(* IEC 61131-3 sources: myCodes/Stone/07.02.2022 - OOPs Approach/MPx_One_New/Mpx_One_Source_Code/MPx_One/3. USHPXMPX010A1/USHPXMPX010A1/[8c990d04-4ef8-4ca1-9757-e845a4517aeb]/Application (part 2) *)

(* ---- 060_MainRegMng.st ---- *)
USING Libs.Logics;
USING System.Timer;
USING System;
USING System.Math;
USING System.Util;

// Uncomment to enable day/night logging
//{DEFINE DNLOGS 1}

VAR_GLOBAL
    MstTempRegStatus : BOOL;
END_VAR

NAMESPACE LibraryNamespaceAndVersion

PROGRAM MainRegMng
    VAR

        TP_s_Timed : TP;
        EEVStartSR : SR;

        CleanRF : RF_TRIG;
        CleanTON : TON;
        //CleanTON_R_Trig : R_TRIG;

        //ContStatusRT : R_TRIG;

        DoorTON : TON;
        DoorLigthTON : TON;
        //DoorOnUsed, DoorOffUsed : FctIsUsed;

        DayNightTrigger, CurtainTrigger : RF_TRIG;//, OnOffDinTrigger : RFTrig;
        DayNightScheduler : MPXScheduler;

        StandbyTON, AndTimeoutTON, AlarmONTON, AlarmTON : TON;
        ContCycle_Pulse : TP;
        StandBy_DIN_R_TRIG : R_TRIG;
        Standby_RS : RS;

        DutySetON, DutySetOFF : TON;

        // Generic function
        AlarmFct : ARRAY [1..1] OF libs.GenericFunctionMng.GenFct_Alarm;
        StageFct : ARRAY [1..1] OF Libs.GenericFunctionMng.GenFct_Stage;
        {IF NOT DEF(MPXONE_BASIC)}
        ModulFct : ARRAY [1..1] OF libs.GenericFunctionMng.GenFct_Modulating;
        {ENDIF}

        TempRegHyst_Left, TempRegHyst_Left2 : REAL;
        TempRegHyst_Right, TempRegHyst_Right2 : REAL;
        //SetP_On, SetP_On2 : REAL;
        //SetP_Off, SetP_Off2 : REAL;

        F_EDGE_firstCycle : F_EDGE;
        FirstCicle_L_Trig   : F_TRIG;

    END_VAR

    VAR_TEMP
        //tmpTempSetP_Offs, tmpTempSetP_Offs2 : REAL;
        AirOffBroken_Delta, AirOnBroken_Delta : REAL;
        EEVOpenOk : BOOL;
        i : DINT;
        //tmpDefCondition : BOOL;
        CompFanDelay_TIME : TIME;

        AlarmTime : TIME;
    END_VAR

    //wait restore default
    IF SW_Update THEN
        RETURN;
    END_IF;

    {REGION STARTUP DELAY}
    // Following regulation will be enabled after the startup delay
    F_EDGE_firstCycle(In := firstCycle);
    FirstCicle_L_Trig(CLK := firstCycle);   // TRAC #115: Stop regoulation at startup (first cycle) in case of startup defrost set
    IF firstCycle OR (FirstCicle_L_Trig.Q AND StartupDef)  THEN
        RETURN;
    END_IF;
    {ENDREGION}

    VirtualProbe := (AnalogInputs.Fct.AirOff * TO_REAL(100 - VirtualComposition) + AnalogInputs.Fct.AirOn * TO_REAL(VirtualComposition)) / 100.0;

    {REGION DAY / NIGHT}
    // Default DayStatus value at startup TRUE

    // Align TOD datatype for APPLICA
    FOR i := LOWER_BOUND(TimeBandStart, 1) TO UPPER_BOUND(TimeBandStart, 1) DO
        ALIGN_TB_TOD(TimeBandStart[i]);
    END_FOR;
    FOR i := LOWER_BOUND(TimeBandEnd, 1) TO UPPER_BOUND(TimeBandEnd, 1) DO
        ALIGN_TB_TOD(TimeBandEnd[i]);
    END_FOR;

    DayNightScheduler(
        CurrentDT := CurrDateTime, Today := CurrentDoW,
        StartTB := TimeBandStart,
        StopTB := TimeBandEnd);

    IF DayNightScheduler.StartTrigger THEN
        DayStatus := TRUE;
    END_IF;

    IF DayNightScheduler.StopTrigger THEN
        DayStatus := FALSE;
    END_IF;

    // Check the curtain switch input
    CurtainTrigger(CLK := DigitalInputs.Fct.Curtain);
    IF CurtainTrigger.Q THEN
        DayStatus := DigitalInputs.Fct.Curtain;
    END_IF;

    // Light adjustment
    DayNightTrigger(CLK := DayStatus);
    IF DayNightTrigger.Q AND Dout_Cfg.Fct.Light.Ch > 0 THEN
        LightsOn := DayStatus;
    END_IF;

    // Light management when door switch is configured
    IF DoorTrigger.Q AND Dout_Cfg.Fct.Light.Ch > 0 THEN
        IF DigitalInputs.Fct.DoorOn OR DigitalInputs.Fct.DoorOff THEN
            LightsOn := DigitalInputs.Fct.DoorOn OR DigitalInputs.Fct.DoorOff;
        ELSIF LightOnDoorDelay = 0 THEN
            LightsOn := FALSE;
        END_IF;
    END_IF;

    // Door timeout for light mng

    DoorLigthTON(IN := LightsOn AND Dout_Cfg.Fct.Light.Ch > 0 AND
        NOT ((DigitalInputs.Fct.DoorOn AND Din_Cfg.fct.DoorOn.Ch > 0) OR (DigitalInputs.Fct.DoorOff AND Din_Cfg.fct.DoorOff.Ch > 0)),
        PT := TO_TIME(TO_DINT(LightOnDoorDelay) * 60 * 1000));

    IF DoorLigthTON.Q AND (Din_Cfg.fct.DoorOff.Ch > 0 OR Din_Cfg.fct.DoorOn.Ch > 0) THEN
        LightsOn := FALSE;
    END_IF;

    // Master / Slave sync
    IF isMaster THEN
        // Notify the slaves on master light status
        FOR i := 1 TO TO_DINT(SlavesNum) DO
            {IF NOT DEF(MPXONE_BASIC)}
            Slaves[i].myCoilStatus[089] := LightsOn;    // set NetworkLight
            Slaves[i].myCoilStatus[079] := AuxOn;       // set NetworkAux
            {ELSE}
            Slaves[i].myCoilStatus[080] := LightsOn;    // set NetworkLight
            Slaves[i].myCoilStatus[071] := AuxOn;       // set NetworkAux
            {ENDIF}
        END_FOR;
    END_IF;

    // Auxiliary output
    CASE CmdAux OF
        0: AuxOn := FALSE;
        1: AuxOn := DayNightOutput AND DayStatus;
        2: AuxOn := TRUE;
    END_CASE;

    {ENDREGION}
    {REGION TIMER FUNCTION}
    TP_s_Timed(IN := DigitalInputs.Fct.Timed, PT := TO_TIME(TO_UINT(TimerDelay) * 60 * 1000));
    TimedOn := TP_s_Timed.Q;
    {ENDREGION}

    {REGION TEMPERATURE REGULATION}
    // regulation probe selection
    RegProbe := VirtualProbe;

    // Night regulation with return temperature probe
    IF NOT DayStatus AND NightPrbReg THEN
        RegProbe := AnalogInputs.Fct.AirOn;
    END_IF;

    // Check setpoint limits on parameter
    TempSetP := MAX(MinTempSet, TempSetP);
    TempSetP := MIN(MaxTempSet, TempSetP);

    TempSetP2 := MAX(MinTempSet, TempSetP2);
    TempSetP2 := MIN(MaxTempSet, TempSetP2);

   //23/01/2020 Filippo Pizzo - TRAC #99: changed action from trigger to keep forced the unit off by remote off

    // Din remote ON/OFF --> force unit off
//    IF DigitalInputs.Fct.RemoteOff THEN
//        UnitStatus := FALSE;
//    END_IF;
    /*
    OnOffDinTrigger(In := DigitalInputs.Fct.RemoteOff);
    IF OnOffDinTrigger.Out THEN
        UnitStatus := NOT DigitalInputs.Fct.RemoteOff;
    END_IF;
    */

    IF UnitOn AND NOT WaitForUpdate THEN
        // Regulation not in alarm
        IF NOT Alarms.Al.AlExtDin.Info.Active AND (NOT(Alarms.Al.AlDelayExtDin.Info.Active AND AlDinDelay>0)) //TRAC #111: if AlDinDelay (param.DIb) = 0 --> only warning
                AND NOT GenFctAlarm_Serious THEN //ISSUE #35

            {REGION TEMPERATURE REGULATION}
            TempRegHyst_Right := TempSetP;
            TempRegHyst_Left := TempSetP;
            TempRegHyst_Right2 := TempSetP2;
            TempRegHyst_Left2 := TempSetP2;

//            SetP_On := TempSetP;
//            SetP_Off := TempSetP;
//            SetP_On2 := TempSetP2;
//            SetP_Off2 := TempSetP2;

            // Control probe lookup
            IF Ain_Cfg.Fct.AirOn.Ch > 0 AND Ain_Cfg.Fct.AirOn.Ch <= TO_SINT(MAX_AIN_CH) THEN
                AirOnBroken := Alarms.Al.Al_PrbBroken[Ain_Cfg.Fct.AirOn.Ch].Info.Active;
            ELSIF Ain_Cfg.Fct.AirOn.Ch < 0 AND Ain_Cfg.Fct.AirOn.Ch >= -4 THEN
                AirOnBroken := Alarms.Al.Al_SerialInputs[-Ain_Cfg.Fct.AirOn.Ch].Info.Active;
            ELSE
                // Probe not configured
                AirOnBroken := TRUE;
            END_IF;

            IF Ain_Cfg.Fct.AirOff.Ch > 0 AND Ain_Cfg.Fct.AirOff.Ch <= TO_SINT(MAX_AIN_CH) THEN

            AirOffBroken := Alarms.Al.Al_PrbBroken[Ain_Cfg.Fct.AirOff.Ch].Info.Active;
            ELSIF Ain_Cfg.Fct.AirOff.Ch < 0 AND Ain_Cfg.Fct.AirOff.Ch >= -4 THEN
                AirOffBroken := Alarms.Al.Al_SerialInputs[-Ain_Cfg.Fct.AirOff.Ch].Info.Active;
            ELSE
                // Probe not configured
                AirOffBroken := TRUE;
            END_IF;

            // Both probe broken or disconnected or not configured
            DutySettings := AirOffBroken AND AirOnBroken;

            // Probe error compensation for AIR OFF broken
            AirOffBroken_Delta := (PrbErrorOffset *  ((100 - TO_REAL(VirtualComposition)) / 100)) * TO_REAL(AirOffBroken);

            // Probe error compensation for AIR ON broken
            AirOnBroken_Delta := (PrbErrorOffset * (TO_REAL( VirtualComposition) / 100)) * TO_REAL(AirOnBroken);

            IF AirOffBroken THEN
                IF VirtualComposition = 0 THEN
                    DutySettings := TRUE;
                ELSE
                     // Switch on other regulation probe
                    RegProbe := AnalogInputs.Fct.AirOn;
                END_IF;
            END_IF;

            IF AirOnBroken THEN
                IF VirtualComposition = 100 THEN
                    DutySettings := TRUE;
                ELSE
                     // Switch on other regulation probe
                    RegProbe := AnalogInputs.Fct.AirOff;
                END_IF;
            END_IF;

            TempRegHyst_Right := TempRegHyst_Right + AirOffBroken_Delta - AirOnBroken_Delta;
            TempRegHyst_Left := TempRegHyst_Left + AirOffBroken_Delta - AirOnBroken_Delta;

            TempRegHyst_Right2 := TempRegHyst_Right2 + AirOffBroken_Delta - AirOnBroken_Delta;
            TempRegHyst_Left2 := TempRegHyst_Left2 + AirOffBroken_Delta - AirOnBroken_Delta;

            IF TempCtrl_DirRev THEN
                                //Standard regulation + Day/Night delta + Smoothline offset + Probe broken offset
                TempRegHyst_Right := TempRegHyst_Right - (SetpNightOffset * TO_REAL( NOT DayStatus ))
                            + (SmLineTempOffset * TO_REAL(EnSmoothLine));
                TempRegHyst_Left := TempRegHyst_Left - TempDiff - (SetpNightOffset * TO_REAL(NOT DayStatus));

                TempRegHyst_Right2 := TempRegHyst_Right2- (SetpNightOffset * TO_REAL( NOT DayStatus ))
                            + (SmLineTempOffset * TO_REAL(EnSmoothLine));

                TempRegHyst_Left2 := TempRegHyst_Left2 - TempDiff2  - (SetpNightOffset * TO_REAL( NOT DayStatus ));

                // Update BMS variables
                ActualTempSetpoint := TempRegHyst_Right;
                ActualTemp2Setpoint := TempRegHyst_Right2;
            ELSE
                //Standard regulation + Day/Night delta + Smoothline offset + Probe broken offset
                TempRegHyst_Right := TempRegHyst_Right + TempDiff + (SetpNightOffset * TO_REAL(NOT DayStatus));
                TempRegHyst_Left := TempRegHyst_Left + (SetpNightOffset * TO_REAL( NOT DayStatus ))
                            - (SmLineTempOffset * TO_REAL(EnSmoothLine));

                TempRegHyst_Right2 := TempRegHyst_Right2 + TempDiff2  + (SetpNightOffset * TO_REAL( NOT DayStatus ));
                TempRegHyst_Left2 := TempRegHyst_Left2 + (SetpNightOffset * TO_REAL( NOT DayStatus ))
                            - (SmLineTempOffset * TO_REAL(EnSmoothLine));

                // Update BMS variables
                ActualTempSetpoint := TempRegHyst_Left;
                ActualTemp2Setpoint := TempRegHyst_Left2;
            END_IF;

            // Double thermostat logic
            IF TempDiff2 > 0.0 THEN

                TempReg(
                	In        := AnalogInputs.Fct.AirOff,
                	SetP      := TempRegHyst_Left,
                	DiffLeft  := 0.0,
                	DiffRight := TempRegHyst_Right - TempRegHyst_Left,
                	Reverse   := TempCtrl_DirRev
                );

                TempReg2(
                	In        := AnalogInputs.Fct.AirOn,
                	SetP      := TempRegHyst_Left2,
                	DiffLeft  := 0.0,
                	DiffRight := TempRegHyst_Right2 - TempRegHyst_Left2,
                	Reverse   := TempCtrl_DirRev
                );
//                TempReg(In := AnalogInputs.Fct.AirOff,
//                    Left := TempRegHyst_Left,
//                    Right := TempRegHyst_Right,
//                    Reverse := TempCtrl_DirRev);

//                TempReg2(In := AnalogInputs.Fct.AirOn,
//                    Left := TempRegHyst_Left2,
//                    Right := TempRegHyst_Right2,
//                    Reverse := TempCtrl_DirRev);

                IF DoubleThermostatConf THEN
                    // OR Condition
                    TempRegStatus := TempReg.Out OR TempReg2.Out;
                    MstTempRegStatus := TempRegStatus;
                ELSE
                    // AND Condition
                    AndTimeoutTON(IN := (TempReg.Out XOR TempReg2.Out) AND DoubleThermSafety > 0, PT := TO_TIME(TO_UINT(DoubleThermSafety) * 60 * 1000));
                        (*Regolation starts if there are request from Sm AND Sr   OR   if there are only one of those AND DoubleThermSafety (dbS) time setted*)
                    TempRegStatus := (TempReg.Out AND TempReg2.Out) OR (AndTimeoutTON.Q AND DoubleThermSafety > 0);
                    MstTempRegStatus := TempRegStatus;
                END_IF;
          ELSE
                TempReg(
                	In        := RegProbe,
                	SetP      := TempRegHyst_Left,
                	DiffLeft  := 0.0,
                	DiffRight := TempRegHyst_Right - TempRegHyst_Left,
                	Reverse   := TempCtrl_DirRev
                );
//                TempReg(In := RegProbe,
//                    Left := TempRegHyst_Left,
//                    Right := TempRegHyst_Right,
//                    Reverse := TempCtrl_DirRev);

                // No double thermostat
                TempRegStatus := TempReg.Out;
                MstTempRegStatus := TempRegStatus;
            END_IF;

            {ENDREGION}

            {REGION CONTINUOUS CYCLE}
            /* Alesssandro Balzan 03/07/2020 changed logic of activation Used TP and added control from disply */

            ContCycle_Pulse(
            	IN := DigitalInputs.Fct.ContCycle OR ManContCycle_byDisplay OR ManContCycle_bySuperv,
            	PT := TO_TIME(TO_DINT(ContCycleTout) * 1000 * 3600)
            );

            IF (DigitalInputs.Fct.ContCycle OR ManContCycle_byDisplay OR ManContCycle_bySuperv) AND ContCycle_Pulse.Q THEN
                ManContinuous := TRUE;
            ELSE
                ContCycle_Pulse(PT := T#0ms); // reset TP
                ManContinuous           := FALSE;
                ManContCycle_byDisplay  := FALSE;
                ManContCycle_bySuperv   := FALSE;
            END_IF;

            //stopped by Alarm
            IF ManContinuous AND ( TempAlarms[1].Low OR TempAlarms[2].Low) AND ContCycleTout > 0 THEN
                ManContinuous           := FALSE;
                ManContCycle_byDisplay  := FALSE;
                ManContCycle_bySuperv   := FALSE;
            END_IF;

            // Defrost priority
            IF ManContinuous AND DfrStatus > DFR_IDLE AND DfrPriorityCont THEN
                ManContinuous           := FALSE;
                ManContCycle_byDisplay  := FALSE;
                ManContCycle_bySuperv   := FALSE;
            END_IF;

            // Keep the regulation active until temperature reach Low temperature alarm threshold
            TempRegStatus := TempRegStatus OR ManContinuous;
            MstTempRegStatus := MstTempRegSTatus OR ManContinuous;

            {ENDREGION}

            {REGION DUTY SETTINGS}
            // Act like a slave for temperature regulation
            IF NOT isMaster AND DutySettings AND NOT Alarms.Al.Al_MA.Info.Active THEN
                TempRegStatus := MstRegStatus;
                RegProbe := MstRegTemp;
                DutySettings := FALSE;
            END_IF;

            IF DutySettings THEN
                DutySetON(IN := NOT DutySetOFF.Q, PT := TO_TIME(TO_DINT(DutySetOnTime) * 60 * 1000));
                DutySetOFF(IN := DutySetON.Q, PT := T#15m);

                TempRegStatus := NOT DutySetON.Q AND NOT DutySetOFF.Q;

                TempRegStatus := TempRegStatus AND DutySetOnTime > 0;

            END_IF;

            // Regulation alarm trigger
            Alarms.Al.Al_Reg.Info.Trigger := DutySettings;
            {ENDREGION}

            {REGION DOOR MANAGEMENT}
            /*DoorOnUsed(FunctionValue := DIN_DOOR_INDEX, Fct := DinFct);
            DoorOffUsed(FunctionValue := DIN_DOOR_ON_INDEX, Fct := DinFct);*/

            DoorTrigger(CLK := DigitalInputs.Fct.DoorOff OR DigitalInputs.Fct.DoorOn);

            Alarms.Al.Warn_Door.Info.Trigger := DigitalInputs.Fct.DoorOff OR DigitalInputs.Fct.DoorOn;

            DoorTON(IN := DigitalInputs.Fct.DoorOff OR DigitalInputs.Fct.DoorOn, PT := TO_TIME(TO_DINT(HighTempBypDoor) * 60 * 1000));
            Alarms.Al.Al_Door.Info.Trigger := DoorTON.Q;

            IF DigitalInputs.Fct.DoorOff AND NOT DoorTON.Q THEN
                TempRegStatus := FALSE;
            END_IF;

//            {IF NOT DEF(MPXONE_BASIC)}
//            myVarTest := FALSE;
//            {ENDIF}

            {ENDREGION}

            {REGION STANDBY}
            StandBy_DIN_R_TRIG(CLK := DigitalInputs.Fct.Standby);
            Standby_RS(S := StandBy_DIN_R_TRIG.Q,
                        R1 := StartupTimeTON.ET > T#0ms OR NOT DigitalInputs.Fct.Standby OR StbyTout = 0);

            Alarms.Al.Status_Standby.Info.Trigger := Standby_RS.Q1 AND NOT StandbyTON.Q;
            StandbyTON(IN := Standby_RS.Q1, PT := TO_TIME(TO_DINT(StbyTout) * 60 * 1000));
            IF Standby_RS.Q1 AND NOT StandbyTON.Q AND StbyTout > 0 THEN
                TempRegStatus := FALSE;
            END_IF;

            {ENDREGION}

            {REGION CLEAN STATUS}
            Alarms.Al.Status_Clean.Info.Trigger := ManClean AND NOT CleanTON.Q;

            CleanRF(CLK := DigitalInputs.Fct.Clean);
            IF CleanRF.Q THEN
                ManClean := DigitalInputs.Fct.Clean;
            END_IF;

            CleanTON(IN := ManClean AND CleanTout > 0, PT := TO_TIME(TO_UDINT(CleanTout) * 60 * 1000));
            IF ManClean AND NOT CleanTON.Q THEN
                TempRegStatus := FALSE;
            END_IF;

            IF (CleanTout > 0 AND CleanTON.ET >= TO_TIME(TO_UDINT(CleanTout) * 60 * 1000)) THEN
                ManClean := FALSE;
            END_IF;

            {ENDREGION}

            // Stop regulation with Natural defrost by running time,
            IF DfrNatural OR DfrCompOff OR           // with compressor=off and defrost until post dripping Ticket TRAC 115)
                (NOT(CompOn) AND DfrStatus>DFR_IDLE AND DfrStatus<DFR_POST_DRIPPING AND DfrType<>1 AND DfrType<>3) THEN

                TempRegStatus := FALSE;

                // Added for hotgas: compON = ON during defrost (not dripping) Independently from request
            ELSIF (DfrType=1 OR DfrType=3) AND DfrStatus>DFR_IDLE AND DfrStatus<DFR_DRIPPING THEN
                TempRegStatus := TRUE;
            END_IF;

            {IF NOT DEF(MPXONE_BASIC)}
            // P10 management
            IF ExvEnCloseLsa AND (Alarms.Al.Al_LSA.Info.Trigger OR Alarms.Al.Al_LSH.Info.Trigger) AND NOT(isMaster AND MstVlvConfig) THEN
                TempRegStatus := FALSE;
//                MstTempRegStatus := FALSE;
            END_IF;
            // PM5 management
            IF ExvEnCloseMOP AND Alarms.Al.Al_MOP.Info.Trigger AND NOT(isMaster AND MstVlvConfig) THEN
                TempRegStatus := FALSE;
//                MstTempRegStatus := FALSE;
            END_IF;
            {ENDIF}

            {REGION Network compressor/solenoid valve output on the Master}
            SlavesTempReq := FALSE;
            // check "TempRegStatus"
            IF isMaster AND SlavesNum > 0 AND MstVlvConfig THEN
                FOR i := 1 TO UPPER_BOUND(Slaves, 1) DO
                    {IF NOT DEF(MPXONE_BASIC)}
                    IF Slaves[i].myInputStatus[87]  THEN
                        SlavesTempReq := TRUE;
                        EXIT;
                    END_IF;
                    {ELSE}
                    IF Slaves[i].myInputStatus[72]  THEN
                        SlavesTempReq := TRUE;
                        EXIT;
                    END_IF;
                    {ENDIF}
                END_FOR;
            END_IF;

            TempRegStatus := TempRegStatus OR SlavesTempReq;
            {ENDREGION}

            {REGION Safety time}
            MinOnT := LIMIT(MinOnT, 0, 15);
            MinOnOnSameT := LIMIT(MinOnOnSameT, 0, 15);
            MinOffT := LIMIT(MinOffT, 0, 15);
            {ENDREGION }

            // Valve has reached the startup opening?
            {IF NOT DEF(MPXONE_BASIC)}
            IF ValveCnf = 6 AND Alarms.Al.Al_Edc.Info.Active THEN
                EEVOpenOk := TRUE;
            ELSE
                EEVOpenOk := (MachineVars.Engine_vars.EEV_vars.CurrentEstimatedPosition > MachineParams.Engine_params.EEV_PARAMS.MinSteps) AND
                            NOT Alarms.Al.Al_Edc.Info.Active;
            END_IF;
            {ELSE}
                EEVOpenOk := TRUE;
            {ENDIF}

            EEVStartSR(
                S1 := TempRegStatus AND (EEVOpenOk OR ValveCnf = 0 OR (isMaster AND SlavesTempReq)),
                R := NOT TempRegStatus
                );

            {REGION Compressor safety times}
            // Comp off during some phase of defrost
            //tmpDefCondition := DfrStatus = DFR_IDLE OR DfrStatus = DFR_POST_DRIPPING ;

            // Allow pump down (NOT AVAILABLE IN CASE OF LIQUID SOLENOID VALVE)
            /*IF DfrPmpDwnDuration > MinOnT THEN
                tmpDefCondition := tmpDefCondition OR DfrStatus = DFR_CALL;
            END_IF;*/

            CntDwnSafT(
                DevReq := EEVStartSR.Q1,
                DevStatus := CompOn,
                MinOnT := MinOnT * 60,
                MinOffT := MinOffT * 60,
                MinOnOnSameT := MinOnOnSameT * 60,
                ResSafT := DfrSafetyTime AND DfrStatus > DFR_CALL,
                DevAlrm := CompAllAlrm,
                En_FB := TRUE

        //        DevOn => BOOL,
        //        FrcdOffByT => ShowCntDwnOff,
        //        FrcdOnByT => ShowCntDwnOn,
        //        CntDwnTSaf => CntDwnT_FrcdOff,
        //        CntDwnTMinOn => CntDwnT_FrcdOn
        //        AbleToOn => BOOL,
        //        AbleToOff => BOOL
                );

            // Function output
            CASE CmdComp OF
                0: // Forced OFF
                    CompOn := FALSE;
                    CompFanDelay_TON(IN := FALSE, PT := T#0ms);
                1: // Automatic
                    IF CompFanDelay > 0 THEN
                        CompFanDelay_TIME := TO_TIME(TO_UDINT(CompFanDelay) * 60 * 1000);
                        CompFanDelay_TON();
                        IF F_EDGE_firstCycle.Out AND CntDwnSafT.DevOn THEN
                            F_EDGE_firstCycle.Reset := TRUE;
                            CompFanDelay_TON(IN := TRUE, PT := CompFanDelay_TIME);
                        ELSIF NOT (CompFanDelay_TON.ET > T#0ms) THEN
                            CompOn := CntDwnSafT.DevOn;
                        ELSIF CompFanDelay_TON.ET >= CompFanDelay_TIME THEN
                            CompFanDelay_TON(IN := FALSE, PT := T#0ms);
                        END_IF;
                    ELSE
                        CompOn := CntDwnSafT.DevOn;
                    END_IF;
                2: // Forced ON
                    CompOn := TRUE;
                    CompFanDelay_TON(IN := FALSE, PT := T#0ms);
            END_CASE;

            // Align slaves about current regulation status
            IF isMaster THEN
                FOR i:=1 TO TO_DINT(SlavesNum) DO
                    {IF NOT DEF(MPXONE_BASIC)}
                    Slaves[i].myCoilStatus[77] := CompOn;   //Set MstRegStatus
                    Slaves[i].myHoldingRegisters[239] := TO_UINT(RegProbe * 10); //Set MstRegTemp
                    {ELSE}
                    Slaves[i].myCoilStatus[069] := CompOn;  //Set MstRegStatus
                    Slaves[i].myHoldingRegisters[178] := TO_UINT(RegProbe * 10); //Set MstRegTemp
                    {ENDIF}
                END_FOR;
            END_IF;
            {ENDREGION }
        ELSE
            // Regulation in alarm with A10 config
            AlarmTime := TO_TIME(TO_REAL(CmpAlConfig) / 100.0 * 15 * 60 * 1000);

            AlarmONTON(IN := NOT AlarmTON.Q, PT := AlarmTime);
            AlarmTON(IN := NOT AlarmTON.Q, PT := T#15m);

            TempRegStatus := NOT AlarmONTON.Q;

            CntDwnSafT(
                DevReq := TempRegStatus,
                DevStatus := CompOn,
                MinOnT := MinOnT * 60,
                MinOffT := MinOffT * 60,
                MinOnOnSameT := MinOnOnSameT * 60,
                ResSafT := FALSE,
                DevAlrm := CompAllAlrm,
                En_FB := TRUE
        //        DevOn => BOOL,
        //        FrcdOffByT => ShowCntDwnOff,
        //        FrcdOnByT => ShowCntDwnOn,
        //        CntDwnTSaf => CntDwnT_FrcdOff,
        //        CntDwnTMinOn => CntDwnT_FrcdOn
        //        AbleToOn => BOOL,
        //        AbleToOff => BOOL
                );

            CompOn := CntDwnSafT.DevOn;
        END_IF;
    ELSE
        // Keep the regulation disabled
        TempReg(
        	In        := -999.9,
        	SetP      := TempSetP,
        	DiffLeft  := 0.0,
        	DiffRight := TempDiff,
        	Reverse   := FALSE
        );

        TempReg2(
        	In        := -999.9,
        	SetP      := TempSetP2,
        	DiffLeft  := 0.0,
        	DiffRight := TempDiff2,
        	Reverse   := FALSE
        );

        TempRegStatus := FALSE;
        CompOn := FALSE;

        //reset Clean Status
        ManClean := FALSE;
        Alarms.Al.Status_Clean.Info.Trigger := FALSE;

        //Keep stand-by status disabled
        Standby_RS(S := FALSE, R1 := TRUE);
        StandBy_DIN_R_TRIG(CLK := TRUE);
        Alarms.Al.Status_Standby.Info.Trigger := FALSE;
    END_IF;
    {ENDREGION}

    {REGION Generic funtions}
    // Staged generic functions
    FOR i:= LOWER_BOUND(GenFctStages_Cfg, 1) TO UPPER_BOUND(GenFctStages_Cfg, 1) DO
        StageFct[i](
        	Stage     := GenFctStages_Cfg[i],
        	EnGenFct  := UnitStatus_WorkingMode = GenFctStages_EnableOn[i] OR
                            (GenFctStages_EnableOn[i] = UNIT_STATUS_GEN_FCT#UNIT_ON AND (UnitStatus_WorkingMode >= UNIT_STATUS_GEN_FCT#DEFROST ) AND (UnitStatus_WorkingMode <= UNIT_STATUS_GEN_FCT#DOOR_OPEN)) OR
//                            (GenFctStages_EnableOn[i] = UNIT_STATUS_GEN_FCT#UNIT_ON AND UnitStatus_WorkingMode = UNIT_STATUS_GEN_FCT#REGULATION_ON) OR
                            GenFctStages_EnableOn[i] = UNIT_STATUS_GEN_FCT#ALWAYS,
        	PrbValues := RegValues
        );

        GenFctStages_Out[i] := StageFct[i].Q;
    END_FOR;

    {IF NOT DEF(MPXONE_BASIC)}
    // Modulating generic functions
    FOR i:= LOWER_BOUND(GenFctModul_Cfg, 1) TO UPPER_BOUND(GenFctModul_Cfg, 1) DO
        ModulFct[i](
        	EnGenFct  := UnitStatus_WorkingMode = GenFctModul_EnableOn[i] OR
                            (GenFctModul_EnableOn[i] = UNIT_STATUS_GEN_FCT#UNIT_ON AND (UnitStatus_WorkingMode >= UNIT_STATUS_GEN_FCT#DEFROST ) AND (UnitStatus_WorkingMode <= UNIT_STATUS_GEN_FCT#DOOR_OPEN)) OR
                            //(GenFctModul_EnableOn[i] = UNIT_STATUS_GEN_FCT#UNIT_ON AND UnitStatus_WorkingMode = UNIT_STATUS_GEN_FCT#REGULATION_ON) OR
                            GenFctModul_EnableOn[i] = UNIT_STATUS_GEN_FCT#ALWAYS,
        	Modul     := GenFctModul_Cfg[i],
        	PrbValues := RegValues
        );

        GenFctModul_Out[i] := ModulFct[i].Q_Modul;
    END_FOR;
    {ENDIF}

    // Alarm generic functions
    GenFctAlarm_Serious := FALSE;
    FOR i:= LOWER_BOUND(GenFctAlarm_Cfg, 1) TO UPPER_BOUND(GenFctAlarm_Cfg, 1) DO
        AlarmFct[i](
            AlarmT          := GenFctAlarm_Cfg[i],
        	EnGenFct        := UnitStatus_WorkingMode = GenFctAlarm_EnableOn[i] OR
                                (GenFctAlarm_EnableOn[i] = UNIT_STATUS_GEN_FCT#UNIT_ON AND (UnitStatus_WorkingMode >= UNIT_STATUS_GEN_FCT#DEFROST ) AND (UnitStatus_WorkingMode <= UNIT_STATUS_GEN_FCT#DOOR_OPEN)) OR
//                                (GenFctAlarm_EnableOn[i] = UNIT_STATUS_GEN_FCT#UNIT_ON AND UnitStatus_WorkingMode = UNIT_STATUS_GEN_FCT#REGULATION_ON) OR
                                GenFctAlarm_EnableOn[i] = UNIT_STATUS_GEN_FCT#ALWAYS,
            PosDinChannel   := Din_Cfg.Fct.GenFctAlrm.Ch,
            ValDinChannel   := DigitalInputs.Fct.GenFctAlrm,
        	PrbValues       := RegValues

        );
        GenFctAlarm_Out[i] := AlarmFct[i].Q;
        IF (GenFctAlarm_Out[i].Hi OR GenFctAlarm_Out[i].Low) AND GenFctAlarm_Out[i].Serious THEN
            GenFctAlarm_Serious := TRUE;
        END_IF;
    END_FOR;
    {ENDREGION}

END_PROGRAM

FUNCTION TimeBandIsToday : BOOL
    VAR_INPUT
        Today : DayOfWeek;
        TimeBandVar : TimeBand;
    END_VAR

    TimeBandIsToday := FALSE;  // Current time band is disabled
    IF TimeBandVar.Day <= 0 THEN
        RETURN;
    END_IF;

    TimeBandIsToday := TimeBandIsToday OR (TimeBandVar.Day = Today OR (TimeBandVar.Day = 7 AND Today = DayOfWeek#Sunday)); // Current time band is only for this day of week
    TimeBandIsToday := TimeBandIsToday OR (TimeBandVar.Day = 8 AND Today >= DayOfWeek#Monday AND Today <= DayOfWeek#Friday); // Current time band is only for monday to friday
    TimeBandIsToday := TimeBandIsToday OR (TimeBandVar.Day = 9 AND Today >= DayOfWeek#Monday); // Current time band is only for monday to saturday
    TimeBandIsToday := TimeBandIsToday OR (TimeBandVar.Day = 10 AND (Today = DayOfWeek#Saturday OR Today = DayOfWeek#Sunday)); // Current time band is only for saturday and sunday
    TimeBandIsToday := TimeBandIsToday OR TimeBandVar.Day = 11; // Current time band is for everyday
END_FUNCTION

FUNCTION TB_TO_INT : INT
    VAR_INPUT
        TimeBandVar : TimeBand;
    END_VAR

    TB_TO_INT := TO_INT(TimeBandVar.Hour) * 60 + TO_INT(TimeBandVar.Minute);

END_FUNCTION

FUNCTION TB_TO_TOD : TOD
    VAR_INPUT
        TimeBandVar : TimeBand;
    END_VAR

    TB_TO_TOD := TO_TOD(TO_DINT(TimeBandVar.Hour) * 3600 + TO_DINT(TimeBandVar.Minute) *60);

END_FUNCTION

FUNCTION TB_TO_TOD_TODAY : TOD
    VAR_INPUT
        TimeBandVar : TimeBand;
        today : DayOfWeek;
    END_VAR

    IF TimeBandIsToday(today, TimeBandVar) THEN
        TB_TO_TOD_TODAY := TB_TO_TOD(TimeBandVar);// TO_TOD(TO_DINT(TimeBandVar.Hour) * 3600 + TO_DINT(TimeBandVar.Minute) * 60);
    ELSE
        TB_TO_TOD_TODAY := TOD#23:59:59;
    END_IF;

END_FUNCTION

FUNCTION ALIGN_TB_TOD
    VAR_IN_OUT
        TimeBandVar : TimeBand;
    END_VAR

    IF TimeBandVar.TimeAPP <> TimeBandVar.MirTimeAPP THEN

        TimeBandVar.Hour := TO_USINT( TO_DINT( TimeBandVar.TimeAPP ) / 3600 );
        TimeBandVar.Minute := TO_USINT( TO_DINT( TimeBandVar.TimeAPP ) / 60 - TO_DINT( TimeBandVar.Hour ) * 60 );

        TimeBandVar.MirTimeAPP := TimeBandVar.TimeAPP;
    ELSE
        TimeBandVar.TimeAPP := TB_TO_TOD( TimeBandVar );
        TimeBandVar.MirTimeAPP := TimeBandVar.TimeAPP;
    END_IF;

END_FUNCTION

FUNCTION ADD_TO_TB : TimeBand
    VAR_INPUT
        tb : TimeBand;
        time : TIME;
    END_VAR
    VAR
        Minutes, Hours : USINT;
        outTb : TimeBand;
    END_VAR

    Hours := TO_USINT(time / (3600 * 1000) );
    Minutes := TO_USINT(time / (60 * 1000) - TO_TIME(TO_DINT(Hours) * 60));

    outTb.Day := tb.Day;
    outTb.Hour := tb.Hour + Hours;
    outTb.Minute := tb.Minute + Minutes;

    // Check time bounds
    IF outTb.Hour > 23 THEN
        outTb.Hour := outTb.Hour - 24;
    END_IF;

    IF outTb.Minute > 59 THEN
        outTb.Minute := outTb.Minute - 60;
    END_IF;

    ADD_TO_TB := outTb;
END_FUNCTION

FUNCTION TBINT_TO_TOD : TOD
    VAR_INPUT
        TimeBandINTVar : INT;
    END_VAR
    VAR
        Minutes, Hours : UINT;
    END_VAR

    Hours := TO_UINT(TimeBandINTVar / 60);
    Minutes := TO_UINT(TimeBandINTVar) - Hours * 60;
    TBINT_TO_TOD := CONCAT_TOD(Hours, Minutes, 0, 0);

END_FUNCTION

FUNCTION_BLOCK MPXScheduler

    VAR_INPUT
        CurrentDT : DATE_AND_TIME;
        Today : DayOfWeek;
    END_VAR

    VAR_IN_OUT
        StartTB : ARRAY [*] OF TimeBand;
        StopTB : ARRAY [*] OF TimeBand;
    END_VAR

    VAR_OUTPUT
        StartTrigger, StopTrigger : BOOL;
        StartIndex : USINT := 0;
    END_VAR

    VAR
        i : DINT;

        now : TOD;
        StartTimeR_TRIG, StopTimeR_TRIG : ARRAY [0..14] OF R_TRIG;

        firstCycle : BOOL := TRUE;
        tmpTOD : TOD;
    END_VAR

    // Get current status from RTC
    now := TO_TOD(CurrentDT);

    // Initial clean of time containers
    StartTrigger := FALSE;
    StopTrigger := FALSE;

    // Check triggers of time bands
    FOR i := LOWER_BOUND(StartTB, 1) TO UPPER_BOUND(StartTB, 1) DO
        tmpTOD := TB_TO_TOD_TODAY(StartTB[i], Today);
        StartTimeR_TRIG[i](CLK := TO_TIME( now - tmpTOD ) < T#5m  AND now > tmpTOD);
        IF StartTimeR_TRIG[i].Q AND NOT firstCycle THEN
            StartTrigger := TRUE;
            StartIndex := TO_USINT(i);
        END_IF;
    END_FOR;
    FOR i := LOWER_BOUND(StopTB, 1) TO UPPER_BOUND(StopTB, 1) DO
        tmpTOD := TB_TO_TOD_TODAY(StopTB[i], Today);
        StopTimeR_TRIG[i](CLK := TO_TIME( now - tmpTOD ) < T#5m AND now > tmpTOD );
        IF StopTimeR_TRIG[i].Q AND NOT firstCycle THEN
            StopTrigger := TRUE;
        END_IF;
    END_FOR;

    firstCycle := FALSE;

END_FUNCTION_BLOCK

FUNCTION_BLOCK MPXSchedulerNew

    VAR_INPUT
        CurrentDT : DATE_AND_TIME;
        Today : DayOfWeek;
    END_VAR

    VAR_IN_OUT
        StartTB : ARRAY [*] OF TimeBand;
        StopTB : ARRAY [*] OF TimeBand;
    END_VAR

    VAR_OUTPUT
        StartTrigger, StopTrigger : BOOL;
        StartIndex : USINT := 0;
    END_VAR

    VAR
        i : DINT;

        now : TOD;
        StartTimeR_TRIG, StopTimeR_TRIG : ARRAY [0..48] OF R_TRIG;

        firstCycle : BOOL := TRUE;
        tmpTOD : TOD;
    END_VAR

    // Get current status from RTC
    now := TO_TOD(CurrentDT);

    // Initial clean of time containers
    StartTrigger := FALSE;
    StopTrigger := FALSE;

    // Check triggers of time bands
    FOR i := LOWER_BOUND(StartTB, 1) TO UPPER_BOUND(StartTB, 1) DO
        tmpTOD := TB_TO_TOD_TODAY(StartTB[i], Today);
        StartTimeR_TRIG[i](CLK := TO_TIME( now - tmpTOD ) < T#5m  AND now > tmpTOD);
        IF StartTimeR_TRIG[i].Q AND NOT firstCycle THEN
            StartTrigger := TRUE;
            StartIndex := TO_USINT(i);
        END_IF;
    END_FOR;
    FOR i := LOWER_BOUND(StopTB, 1) TO UPPER_BOUND(StopTB, 1) DO
        tmpTOD := TB_TO_TOD_TODAY(StopTB[i], Today);
        StopTimeR_TRIG[i](CLK := TO_TIME( now - tmpTOD ) < T#5m AND now > tmpTOD );
        IF StopTimeR_TRIG[i].Q AND NOT firstCycle THEN
            StopTrigger := TRUE;
        END_IF;
    END_FOR;

    firstCycle := FALSE;

END_FUNCTION_BLOCK

END_NAMESPACE

(* ---- 070_DefrostMng.st ---- *)
USING System;
USING Libs.Hysteresis;
USING System.Timer;
USING System.Math;
USING Libs.GenericFunctionMng;

// Uncomment to enable defrost logging
//{DEFINE DEFLOGS 1}

{DEFINE DEFROST_ANALISYS}

{DEFINE DEFROST_TO_SKIP 3}
{DEFINE DEFROST_TO_WAIT 8}

NAMESPACE LibraryNamespaceAndVersion

PROGRAM DfrMng
    VAR
        DfrSched : MPXScheduler;
        Staggered1, Staggered2 : MPXSchedulerNew;
        CallRTRIG, DfrRTRIG : R_TRIG;
        DfrOnTON, DfrOnTON2 : TON;
        DfrDuration, DfrDuration2 : USINT;
        DfrMaxDurationT, DfrMaxDuration2T : UDINT;
        SkipCounter, SkipCounter2 : SINT := 1 - DEFROST_TO_WAIT;
        SkippedCounter : USINT;
        SkipSR : SR;
        MachineTON, startupDefTON : TON;

        startLocal, startNetwork, startupDefSR : SR;
        TempControl, TempControl2 : HysterAdv;

        RunningTTON : TON;
        RunningTTON_2evap : TON;
        SequentialOnTON, SequentialOffTON : TON_PAUSE;
        CurrentTBisPow : BOOL;

        SlaveDfrDelay_TON : TON;

        (**Used by "defrost start by delta" function*)
        DfrStartByDelta_TON : TON;

//      DfrOnTimer : TIME;
//      ForceTON : TON;
//      ForceWrite, ForceValue : BOOL;
//      TBRunningIndex : USINT;
//      tmpYears, tmpMonth, tmpDays, tmpHours, tmpMin, tmpSec, tmpMillis : UINT;
    END_VAR

    VAR_TEMP
        nullTB                          : ARRAY [0..1] OF TimeBand;
        staggeredTB1, staggeredTB2      : ARRAY [0..47] OF TimeBand;
        timeCheckEnd, tempCheckEnd      : BOOL;
        heaterType, hotGasType, multiplexHotGasType : BOOL;
        tempRegDef                      : BOOL;
        i                               : DINT;
        slavesOk                        : BOOL;
        staggeredDelay                  : TIME;
        tmpDfrEndTemp, tmpDfrEnd2Temp   : REAL;
        DfrEndedByTime, Dfr2EndedByTime : BOOL;
        tmpDailyDfrNum, tmpDailyDfrNum2 : USINT(0..48);

        DfrActualInterval_T             : TIME;
        EnProbe1, EnProbe2              : BOOL;
        DfrProbe                        : REAL;
    END_VAR

    //wait restore default
    IF SW_Update THEN
        RETURN;
    END_IF;

    // Following regulation will be enabled after the startup delay
    IF firstCycle THEN

        //SPLIT_DT(CurrDateTime, tmpYears, tmpMonth, tmpDays, tmpHours, tmpMin, tmpSec, tmpMillis);

        // Avoid unexpected defrost at power on
        //DfrStartedDT := CurrDateTime;

        // Startup defrost trigger
        startupDefSR(S1 := StartupDef, R := FALSE);

        RETURN;
    END_IF;

    // Startup defrost
    startupDefSR(S1 := FALSE, R := startupDefTON.Q);
    startupDefTON(IN := startupDefSR.Q1 AND StartupDef, PT := TO_TIME(TO_DINT(DfrPowOnDelay) * 1000 * 60));
    IF startupDefTON.Q AND StartupDef THEN
        ManDfr := TRUE;
        NetworkDfr := isMaster;
//        StartupDef := FALSE;
    END_IF;

    // Align TOD datatype for APPLICA
    FOR i := LOWER_BOUND(DfrStart, 1) TO UPPER_BOUND(DfrStart, 1) DO
        ALIGN_TB_TOD(DfrStart[i]);
    END_FOR;

    // Call the scheduler
    DfrSched(
        CurrentDT := CurrDateTime, Today := CurrentDoW,
        StartTB := DfrStart, StopTB := nullTB);

    // Staggered defrost

    CASE DailyDfrNum OF //calculate the number of defrost events
            1..12:  tmpDailyDfrNum := DailyDfrNum;
            13 :    tmpDailyDfrNum := 24;
            14 :    tmpDailyDfrNum := 48;
    END_CASE;

    //tmpDailyDfrNum := DailyDfrNum;
    //DailyDfrNum := tmpDailyDfrNum;

    IF tmpDailyDfrNum > 0 THEN
        CASE tmpDailyDfrNum OF
            1..12: staggeredDelay := T#24h / tmpDailyDfrNum;
            24 : staggeredDelay := T#1h;
            48 : staggeredDelay := T#30m;
        END_CASE;

        FOR i := 0 TO TO_DINT(tmpDailyDfrNum - 1) DO
            staggeredTB1[i] := ADD_TO_TB(DfrStart[1], staggeredDelay * (i + 1) );
        END_FOR;

        Staggered1(CurrentDT := CurrDateTime, Today := CurrentDoW,
            StartTB := staggeredTB1, StopTB := nullTB);
    END_IF;

    //tmpDailyDfrNum2 := DailyDfrNum2;
    //DailyDfrNum2 := tmpDailyDfrNum2;

    CASE DailyDfrNum2 OF //calculate the number of defrost events
            1..12:  tmpDailyDfrNum2 := DailyDfrNum2;
            13 :    tmpDailyDfrNum2 := 24;
            14 :    tmpDailyDfrNum := 48;
    END_CASE;

    IF tmpDailyDfrNum2 > 0 THEN
        CASE DailyDfrNum2 OF
            1..12: staggeredDelay := T#24h / tmpDailyDfrNum2;
            24 : staggeredDelay := T#1h;
            48 : staggeredDelay := T#30m;
        END_CASE;

        FOR i := 0 TO TO_DINT(tmpDailyDfrNum2 - 1) DO
            staggeredTB2[i] := ADD_TO_TB(DfrStart[2], staggeredDelay * (i + 1) );
        END_FOR;

        Staggered2(CurrentDT := CurrDateTime, Today := CurrentDoW,
            StartTB := staggeredTB2, StopTB := nullTB);
    END_IF;

    // Running time defrost
    IF Ain_Cfg.Fct.Defrost.ch > 0 THEN
        RunningTTON(IN := AnalogInputs.Fct.Defrost < DfrTempRun AND NOT (DfrStatus > DFR_IDLE) AND DfrTimeRun > 0 AND NOT Alarms.Al.Al_PrbBroken[Ain_Cfg.Fct.Defrost.ch].Info.Active,
                    PT := TO_TIME(TO_DINT(DfrTimeRun) * 1000 * 60));
        IF RunningTTON.Q THEN
            ManDfr := TRUE;
        END_IF;
    END_IF;

    // Running time defrost evaporator 2
    IF Ain_Cfg.Fct.Defrost2.ch > 0 THEN
        RunningTTON_2evap(IN := AnalogInputs.Fct.Defrost2 < DfrTempRun AND NOT (DfrStatus > DFR_IDLE) AND DfrTimeRun > 0 AND NOT Alarms.Al.Al_PrbBroken[Ain_Cfg.Fct.Defrost2.ch].Info.Active,
                            PT := TO_TIME(TO_DINT(DfrTimeRun) * 1000 * 60));
        IF RunningTTON_2evap.Q THEN
            ManDfr := TRUE;
        END_IF;
    END_IF;

    {REGION DEFROST START BY DELTA}
    //  (issue #16) ------------------------------------------------
    IF  DfrStartByDeltaThrsh>0 AND DfrStartByDeltaPrb1 > 0 AND DfrStartByDeltaPrb2 > 0 THEN
        IF TO_USINT(DfrStartByDeltaPrb1) <= AIN_NUM THEN //real probe
                // Probe 1 is correctly configured and not in Alarm
            IF  (Ain_Cfg.Arr[DfrStartByDeltaPrb1].Ch>0 AND Ain_Cfg.Arr[DfrStartByDeltaPrb1].Ch <= TO_SINT(MAX_AIN_CH) AND
                NOT Alarms.Al.Al_PrbBroken[Ain_Cfg.Arr[DfrStartByDeltaPrb1].Ch].Info.Active) THEN
                EnProbe1 := TRUE;
            END_IF;
        ELSE
            EnProbe1 := TRUE;  // virtual or calculated probe
        END_IF;

        IF TO_USINT(DfrStartByDeltaPrb2) <= AIN_NUM THEN //real probe
                 // Probe 2 is correctly configured and not in Alarm
            IF (Ain_Cfg.Arr[DfrStartByDeltaPrb2].Ch>0 AND Ain_Cfg.Arr[DfrStartByDeltaPrb2].Ch <= TO_SINT(MAX_AIN_CH) AND
                NOT Alarms.Al.Al_PrbBroken[Ain_Cfg.Arr[DfrStartByDeltaPrb2].Ch].Info.Active) THEN
                EnProbe2 := TRUE;
            END_IF;
        ELSE
            EnProbe2 := TRUE;  // virtual or calculated probe
        END_IF;

        DfrStartByDelta_TON(
            IN := DfrStatus=DFR_IDLE AND // If not defrosting right now,
                EnProbe1 AND EnProbe2 AND
                RegValues[DfrStartByDeltaPrb1]-RegValues[DfrStartByDeltaPrb2] > DfrStartByDeltaThrsh, // Difference is greather than threshold
            PT := TO_TIME(TO_DINT(DfrStartByDeltaT)*60*1000)
        );
        IF DfrStartByDelta_TON.Q THEN
            ManDfr := TRUE;
        END_IF;
    ELSE
        DfrStartByDelta_TON(IN := FALSE, PT := T#0s);
    END_IF;

    {ENDREGION}

    // Sequential stop defrost
    SequentialOffTON(IN := UnitOn AND NOT SequentialOffTON.Q AND NOT SequentialOnTON.Q,
                    PT := TO_TIME(TO_DINT(DfrOffTimeSeq) * 1000 * 60), PAUSE := CompOn);
    SequentialOnTON(IN := UnitOn AND NOT SequentialOffTON.Q AND NOT SequentialOnTON.Q,
                    PT := TO_TIME(TO_DINT(DfrOnTimeSeq) * 1000 * 60), PAUSE := NOT CompOn);

    IF SequentialOnTON.Q AND (DfrOffTimeSeq > 0) THEN
        DfrNatural := TRUE;
    END_IF;
    IF SequentialOffTON.Q AND DfrNatural THEN
        DfrNatural := FALSE;
    END_IF;

    // Reset defrost if finished manually
    IF DfrStatus > DFR_IDLE AND NOT ManDfr AND startLocal.Q1 THEN
        DfrStatus := DFR_IDLE;
        ManDfr := FALSE;
        //Allows to stop the Defrost on the slave
        IF NOT isMaster THEN
            NetworkDfr := FALSE;
        END_IF;
        DfrOnTON(IN := FALSE, PT := T#0s);
        DfrOnTON2(IN := FALSE, PT := T#0s);
        {IF DEF(MPXONE_MEDIUM)}
        MachineVars.ManualPositioner_vars.ManualPositioningEnable := FALSE;
        {ENDIF}
    END_IF;

    // Finish defrost by the Disable of DI or Unit off
    IF DfrStatus > DFR_IDLE AND (DigitalInputs.Fct.EnDfr OR NOT UnitOn OR DigitalInputs.Fct.DefrostMirror) THEN //TRAC #120 stop defrost by "dir" input

        IF DigitalInputs.Fct.EnDfr THEN // If defrost is disabled by digital input  book a new defrost waiting for the re-enable
        DfrBook := TRUE;
        END_IF;

        DfrStatus := DFR_IDLE;
        ManDfr := FALSE;
        NetworkDfr := FALSE;
        DfrOnTON(IN := FALSE, PT := T#0s);
        DfrOnTON2(IN := FALSE, PT := T#0s);
        {IF DEF(MPXONE_MEDIUM)}
        MachineVars.ManualPositioner_vars.ManualPositioningEnable := FALSE;
        {ENDIF}
    END_IF;

    // Also if i'm the slave and is manually ended on master stop the local defrost
    // and if the master stop the network
    IF DfrStatus > DFR_IDLE AND NOT NetworkDfr AND startNetwork.Q1 THEN
        DfrStatus := DFR_IDLE;
        ManDfr := FALSE;
        DfrOnTON(IN := FALSE, PT := T#0s);
        DfrOnTON2(IN := FALSE, PT := T#0s);
        {IF DEF(MPXONE_MEDIUM)}
        MachineVars.ManualPositioner_vars.ManualPositioningEnable := FALSE;
        {ENDIF}

        // Notify the slave to stop the defrost
        IF isMaster AND NOT DisNetworkDfr AND SlavesNum > 0 THEN
            FOR i := 1 TO TO_DINT(SlavesNum) DO
                {IF NOT DEF(MPXONE_BASIC)}
                Slaves[i].myCoilStatus[059] := FALSE; // ManDfr in BMS table ManDfr
                {ELSE}
                Slaves[i].myCoilStatus[053] := FALSE; // ManDfr in BMS table ManDfr
                {ENDIF}
                Slaves[i].myCoilStatus[029] := FALSE; // Reset network Defrost
            END_FOR;
        END_IF;
        //ForceWrite := TRUE;
        //ForceValue := FALSE;
    END_IF;

    // In case of network and a manual stop of the local only
    IF DfrStatus > DFR_IDLE AND NOT ManDfr AND startNetwork.Q1 THEN
        DfrStatus := DFR_IDLE;
        ManDfr := FALSE;
        NetworkDfr := FALSE;
        DfrOnTON(IN := FALSE, PT := T#0s);
        DfrOnTON2(IN := FALSE, PT := T#0s);
        {IF DEF(MPXONE_MEDIUM)}
        MachineVars.ManualPositioner_vars.ManualPositioningEnable := FALSE;
        {ENDIF}
    END_IF;

    // Start cause memory reset on IDLE
    startLocal(S1 := FALSE, R := DfrStatus = DFR_IDLE);
    startNetwork(S1 := FALSE, R := DfrStatus = DFR_IDLE);

    // Check the configuration
    CASE DfrType OF
        0: // HEATER BY TEMPERATURE
        // Defrost end condition
        timeCheckEnd := TRUE; tempCheckEnd := TRUE;
        // Type of defrost
        heaterType := TRUE; hotGasType := FALSE; multiplexHotGasType := FALSE;
        1: // HOT GAS BY TEMPERATURE
        // Defrost end condition
        timeCheckEnd := TRUE; tempCheckEnd := TRUE;
        // Type of defrost
        heaterType := FALSE; hotGasType := TRUE; multiplexHotGasType := FALSE;
        2: // heater by time
        // Defrost end condition
        timeCheckEnd := TRUE; tempCheckEnd := FALSE;
        // Type of defrost
        heaterType := TRUE; hotGasType := FALSE; multiplexHotGasType := FALSE;
        3: // hot gas by time
        // Defrost end condition
        timeCheckEnd := TRUE; tempCheckEnd := FALSE;
        // Type of defrost
        heaterType := FALSE; hotGasType := TRUE; multiplexHotGasType := FALSE;
        4: // heater by time with temp. control
        // Defrost end condition
        timeCheckEnd := TRUE; tempCheckEnd := FALSE;
        // Type of defrost
        heaterType := TRUE; hotGasType := FALSE; multiplexHotGasType := FALSE;
        tempRegDef := TRUE;
        5: // multiplexed hot gas by temperature
        // Defrost end condition
        timeCheckEnd := TRUE; tempCheckEnd := TRUE;
        // Type of defrost
        heaterType := FALSE; hotGasType := FALSE; multiplexHotGasType := TRUE;
        6: // multiplexed hot gas by time
        // Defrost end condition
        timeCheckEnd := TRUE; tempCheckEnd := FALSE;
        // Type of defrost
        heaterType := FALSE; hotGasType := FALSE; multiplexHotGasType := TRUE;
    END_CASE;

    // Defrost alarm management
    IF Alarms.Al.AlExtDin.Info.Active OR (Alarms.Al.AlDelayExtDin.Info.Active AND AlDinDelay>0)   //TRAC #111: if AlDinDelay (param.DIb) = 0 --> only warning
            OR GenFctAlarm_Serious THEN //ISSUE #35
        DfrStatus := DFR_IDLE;
        ManDfr := FALSE;
        NetworkDfr := FALSE;
    END_IF;

    // Master controller align status of slaves: used for defrost can end in the slaves
    IF isMaster AND SlavesNum > 0 THEN
        FOR i := 1 TO TO_DINT(SlavesNum) DO
            {IF NOT DEF(MPXONE_BASIC)}
            Slaves[i].myHoldingRegisters[212] := TO_UINT(DfrStatus); // DfrMstStatus in BMS table
            {ELSE}
            Slaves[i].myHoldingRegisters[166] := TO_UINT(DfrStatus); // DfrMstStatus in BMS table
            {ENDIF}
        END_FOR;
    END_IF;

    // Multiplexed defrost on offline slave with safety
    DfrHotGasSafetyActive := Alarms.Al.Al_MA.Info.Active AND DfrStatus > DFR_IDLE AND DfrHotGasSafety;

    //Logs Info
    DfrInProgress := DfrStatus > DFR_IDLE;

    // Defrost request by digital input- TRAC #89
    IF Din_Cfg.Fct.CallDfr.Ch <> 0 THEN
        CallRTRIG(CLK := NOT( DigitalInputs.Fct.CallDfr) AND NOT(DigitalInputs.Fct.EnDfr)); //TRAC #120 acivate defrost by "Dir" input
    ELSE
        CallRTRIG(CLK := FALSE);
    END_IF;

    CASE DfrStatus OF
        DFR_IDLE : //------------- DEFROST IDLE STATUS

            // Conditions to start Dfr

            // Check if configured DI allow a Dfr
            IF NOT DigitalInputs.Fct.EnDfr AND UnitOn  THEN

                // Call Defrost by digital input
                IF CallRTRIG.Q OR DfrBook OR (Din_Cfg.Fct.DefrostMirror.Ch>0 AND NOT DigitalInputs.Fct.DefrostMirror) THEN //start defrost by digital input of by re-enable - TRAC #89 #120
                    DfrStatus := DFR_CALL;
                    DfrBook := FALSE;
                END_IF;

                // Schedulers
                IF DfrSched.StartTrigger AND NOT Alarms.Al.Al_RTC.Info.Active THEN
                    DfrStatus := DFR_CALL;
                    IF DfrSched.StartIndex >= TO_USINT(LOWER_BOUND(PowDfrConf, 1)) AND DfrSched.StartIndex <= TO_USINT(LOWER_BOUND(PowDfrConf, 1)) THEN
                        CurrentTBisPow := PowDfrConf[DfrSched.StartIndex];
                    ELSE
                        CurrentTBisPow := FALSE;
                    END_IF;
                END_IF;
                IF Staggered1.StartTrigger THEN
                    DfrStatus := DFR_CALL;
                    CurrentTBisPow := PowDfrConf[1];
                END_IF;
                IF Staggered2.StartTrigger THEN
                    DfrStatus := DFR_CALL;
                    CurrentTBisPow := PowDfrConf[2];
                END_IF;

                // Power defrost on night
                CurrentTBisPow := CurrentTBisPow OR NOT DayStatus;

                // Maximum time between Dfr start
                DfrActualInterval_T := CurrDateTime - DfrStartedDT;
                IF (DfrInterval > 0) AND DfrActualInterval_T >= TO_TIME(TO_DINT(DfrInterval) * 1000 * 3600) THEN
                    DfrStatus := DFR_CALL;
                END_IF;

                // Only if defrost is called by Inputs, scheduler or DI start a network defrost
                IF isMaster AND DfrStatus = DFR_CALL THEN
                    NetworkDfr := TRUE;
                END_IF;

                // Master call network defrost
                IF NetworkDfr AND NOT DisNetworkDfr THEN
                    DfrStatus := DFR_CALL;
                    startNetwork(S1 := TRUE, R := FALSE);

                    // Notify the slave to start the defrost
                    IF isMaster AND NOT DisNetworkDfr AND SlavesNum > 0 THEN
                        FOR i := 1 TO TO_DINT(SlavesNum) DO
                            Slaves[i].myCoilStatus[29] := TRUE; // NetworkDfr in BMS table
                        END_FOR;
                    END_IF;
                    //ForceWrite := TRUE;
                    //ForceValue := TRUE;
                END_IF;

                // Skip defrost check
                SkipSR(S1 := DfrSkipEn AND (SkipCounter >= DEFROST_TO_SKIP OR SkipCounter2 >= DEFROST_TO_SKIP), R := NOT DfrSkipEn OR SkippedCounter <= 0 );
                IF SkipSR.Q1 AND DfrStatus > DFR_IDLE THEN

                    DfrStatus := DFR_IDLE;
                    SkippedCounter := SkippedCounter + 1;

                    IF SkippedCounter >= DEFROST_TO_SKIP THEN
                        SkipCounter := 1;
                        SkipCounter2 := 1;
                        SkippedCounter := 0;
                    END_IF;

                END_IF;

            END_IF;

            // Always force the DO to off
            DfrOn := FALSE;
            DfrOn2 := FALSE;
            DfrCompOff := FALSE;

            // Reset service timer
            MachineTON(IN := FALSE, PT := T#10s); // Reset TIMER

            IF ManDfr THEN
                DfrStatus := DFR_CALL;
                startLocal(S1 := TRUE, R := FALSE);
            END_IF;

            // Align manual command from SPV or APP
            IF DfrStatus = DFR_CALL THEN
                ManDfr := TRUE;
            END_IF;

            {IF NOT DEF(MPXONE_BASIC)}
            // Multiplexed hot gas normal operating mode
            IF multiplexHotGasType THEN
                // Suction solenoid valve for Multiplexed Hot Gas Defrost
                S_VlvOn := TRUE;
                // Equalizing solenoid valve for Multiplexed Hot Gas Defrost
                E_VlvOn := FALSE;
            ELSE
                S_VlvOn := FALSE;
                E_VlvOn := FALSE;
            END_IF;
            {ENDIF}

        DFR_CALL : //------------- DEFROST CALL STATUS
            {IF NOT DEF(MPXONE_BASIC)}
            IF multiplexHotGasType THEN
                // Suction solenoid valve for Multiplexed Hot Gas Defrost
                S_VlvOn := TRUE;
                // Equalizing solenoid valve for Multiplexed Hot Gas Defrost
                E_VlvOn := FALSE;
            ELSE
                S_VlvOn := FALSE;
                E_VlvOn := FALSE;
            END_IF;
            {ENDIF}

            //Allows to stop local defrost
            IF ManDfr AND NOT isMaster THEN
                startLocal(S1 := TRUE, R := FALSE);
            END_IF;

            // Count PD time
           MachineTON(IN := TRUE, PT := TO_TIME(DfrPmpDwnDuration * 1000)); // Count

            // Defrost start conditions
            DfrStatus := DFR_DFR;
            // Safety conditions to start Dfr (Timing)
            IF ( CompOn AND multiplexHotGasType ) OR NOT MachineTON.Q THEN
                DfrStatus := DFR_CALL;
            END_IF;
            // Continuous cycle
            IF ManContinuous AND NOT DfrPriorityCont THEN
                DfrStatus := DFR_CALL;
            END_IF;
            // Compressor timing
            IF NOT DfrSafetyTime AND CntDwnSafT.DevOn AND NOT CntDwnSafT.AbleToOff THEN
                 DfrStatus := DFR_CALL;
            END_IF;

            IF NOT isMaster AND DfrPowOnDelay > 0 AND NetworkDfr THEN
                SlaveDfrDelay_TON(IN := TRUE, PT := TO_TIME(TO_UDINT(DfrPowOnDelay) * 60 * 1000));
                IF NOT  SlaveDfrDelay_TON.Q THEN
                    DfrStatus := DFR_CALL;
                ELSE
                    SlaveDfrDelay_TON(IN := FALSE, PT := T#0s);
                    DfrStatus := DFR_DFR;
                END_IF;
            END_IF;

            // Defrost will start next execution
            IF DfrStatus = DFR_DFR THEN
                // Perform the Dfr action
                DfrCompOff := heaterType OR multiplexHotGasType;

                DfrOn := timeCheckEnd;
                DfrOn2 := Ain_Cfg.Fct.Defrost2.ch > 0;
////                DfrOn := DoutChannels[7] > 0;
////                DfrOn2 := DoutChannels[8] > 0;
            END_IF;

        DFR_DFR : //------------- DEFROST ON STATUS

            {IF NOT DEF(MPXONE_BASIC)}
            IF multiplexHotGasType THEN
                // Suction solenoid valve for Multiplexed Hot Gas Defrost
                S_VlvOn := FALSE;
                // Equalizing solenoid valve for Multiplexed Hot Gas Defrost
                E_VlvOn := FALSE;
            ELSE
                S_VlvOn := FALSE;
                E_VlvOn := FALSE;
            END_IF;

//            IF DfrType = 1 OR DfrType = 3 THEN
//                TempRegStatus := TRUE;
//            END_IF;
            {ENDIF}

            // Timer to count Dfr duration
            DfrRTRIG(CLK := TRUE);
            IF DfrRTRIG.Q THEN
                LibraryNamespaceAndVersion.SetLastDfrTime_RTC_MEM(CurrDateTime);
            END_IF;

            //DfrOnTimer := CurrDateTime - DfrStartedDT;
            DfrMaxDurationT := TO_UDINT(DfrMaxDuration + DfrPowTime * TO_USINT(CurrentTBisPow)) * 1000 * 60;
            DfrOnTON(
            	IN := TRUE,
            	PT := TO_TIME(DfrMaxDurationT)
            );
            DfrMaxDuration2T := TO_UDINT(DfrMaxDuration2 + DfrPowTime * TO_USINT(CurrentTBisPow)) * 1000 * 60;
            DfrOnTON2(
            	IN := TRUE,
            	PT := TO_TIME(DfrMaxDuration2T)
            );

            // BY TIME
            //IF DfrOnTimer >= TO_TIME(TO_DINT(DfrMaxDuration) * 1000 * 60) AND DfrOn AND timeCheckEnd AND DoutChannels[7] > 0 THEN // Convert minutes UINT to TIME
            IF DfrOnTON.Q AND (DfrOn OR DfrType = 4) AND timeCheckEnd THEN //AND PrbChannels[2] > 0 DoutChannels[7] > 0 THEN
                DfrOn := FALSE;
                DfrEndedByTime := TRUE;
                //DfrStatus := DFR_CHECK_END;
                IF tempRegDef AND (Dfr2EndedByTime OR (Ain_Cfg.Fct.Defrost2.ch = 0)) THEN
                    DfrStatus := DFR_CHECK_END;
                END_IF;

                // Signal end by timeout
                IF tempCheckEnd AND DfrEndAlTimeout THEN
                    Alarms.Al.DfrTout1.Info.Trigger := TRUE;
                END_IF;
            END_IF;

            // BY TIME EVAPORATOR 2
            //IF DfrOnTimer >= TO_TIME(TO_DINT(DfrMaxDuration2) * 1000 * 60) AND DfrOn2 AND timeCheckEnd AND DoutChannels[8] > 0 THEN // Convert minutes UINT to TIME
            IF DfrOnTON2.Q AND (DfrOn2 OR DfrType = 4) AND timeCheckEnd THEN //AND PrbChannels[6] > 0 DoutChannels[8] > 0 THEN
                DfrOn2 := FALSE;
                Dfr2EndedByTime := TRUE;
                //DfrStatus := DFR_CHECK_END;
                IF tempRegDef AND (DfrEndedByTime  OR (Ain_Cfg.Fct.Defrost.ch = 0)) THEN
                    DfrStatus := DFR_CHECK_END;
                END_IF;

                // Signal end by timeout
                IF tempCheckEnd AND DfrEndAlTimeout THEN
                    Alarms.Al.DfrTout2.Info.Trigger := TRUE;
                END_IF;
            END_IF;

            // BY TEMPERATURE

            // Power Defrost offset
            tmpDfrEndTemp := DfrEndTemp + DfrPowTemp * TO_REAL(CurrentTBisPow);
            tmpDfrEnd2Temp := DfrEnd2Temp + DfrPowTemp * TO_REAL(CurrentTBisPow);

            IF (AnalogInputs.Fct.Defrost > tmpDfrEndTemp AND Ain_Cfg.Fct.Defrost.ch > 0
                AND Ain_Cfg.Fct.Defrost.ch <= MAX_AIN_CH
                AND NOT Alarms.Al.Al_PrbBroken[Ain_Cfg.Fct.Defrost.ch].Info.Active) AND
                DfrOn AND tempCheckEnd THEN //DoutChannels[7] > 0 THEN

                DfrOn := FALSE;
                // Reset timeout
                Alarms.Al.DfrTout1.Info.Trigger := FALSE;
                //DfrStatus := DFR_CHECK_END;

                // Skip defrost counter check
                DfrDuration := TO_USINT(TO_REAL(DfrOnTON.ET) / TO_REAL(DfrMaxDurationT) * 100.0);
                IF DfrDuration < DfrSkipDuration AND DfrSkipEn THEN
                    SkipCounter := SkipCounter + 1;
                END_IF;

            END_IF;

            // BY TEMPERATURE EVAPORATOR 2
            IF (AnalogInputs.Fct.Defrost2 > tmpDfrEnd2Temp AND Ain_Cfg.Fct.Defrost2.ch > 0
                AND Ain_Cfg.Fct.Defrost.ch <= MAX_AIN_CH
                AND NOT Alarms.Al.Al_PrbBroken[Ain_Cfg.Fct.Defrost2.ch].Info.Active) AND
                DfrOn2 AND tempCheckEnd THEN //DoutChannels[8] > 0 THEN

                DfrOn2 := FALSE;
                // Reset timeout
                Alarms.Al.DfrTout2.Info.Trigger := FALSE;
                //DfrStatus := DFR_CHECK_END;

                // Skip defrost counter check
                DfrDuration2 := TO_USINT(TO_REAL(DfrOnTON2.ET) / TO_REAL(DfrMaxDuration2T) * 100.0);
                IF DfrDuration2 < DfrSkipDuration AND DfrSkipEn THEN
                    SkipCounter2 := SkipCounter2 + 1;
                END_IF;

            END_IF;

            // Finish the defrost on unconfigured evaporators DO (won't work anyway)
//            IF NOT (PrbChannels[2] > 0) AND tempCheckEnd THEN //(DoutChannels[7] > 0) THEN
//                DfrOn := FALSE;
//            END_IF;
//            IF NOT (PrbChannels[6] > 0) AND tempCheckEnd THEN //(DoutChannels[8] > 0) THEN
//                DfrOn2 := FALSE;
//            END_IF;

            // Temperature regulation
            IF tempRegDef AND Ain_Cfg.Fct.Defrost.ch > 0 AND NOT DfrEndedByTime THEN
                TempControl(
                	In      := AnalogInputs.Fct.Defrost,
                	SetP      := tmpDfrEndTemp,
                	DiffLeft  := 1.0,
                	DiffRight := 0.0,
                	Reverse   := TRUE,
                    Out       => DfrOn
                );
            END_IF;

            IF tempRegDef AND  Ain_Cfg.Fct.Defrost2.ch > 0 AND NOT Dfr2EndedByTime THEN
                TempControl2(
                	In      := AnalogInputs.Fct.Defrost2,
                	SetP      := tmpDfrEnd2Temp,
                	DiffLeft  := 1.0,
                	DiffRight := 0.0,
                	Reverse   := TRUE,
                    Out       => DfrOn2
                );
            END_IF;

            // Finish the defrost status only when both evaporators are OK and slaves are ok
            IF NOT tempRegDef AND NOT DfrOn AND NOT DfrOn2 THEN
                DfrStatus := DFR_CHECK_END;
            END_IF;

        DFR_CHECK_END : //------------- DEFROST CHECK END CONDITIONS STATUS

            DfrCompOff := TRUE;
            // Wait for other controllers on the network
            DfrOn := FALSE;
            DfrOn2 := FALSE;

            // Get feedback for slaves defrost status
            IF NOT isMaster THEN
                // Slaves controllers can finish + check if master was not in sync
                slavesOk := DfrMstStatus > DFR_CHECK_END OR DfrMstStatus <= DFR_IDLE OR NOT DfrMasterEndSync OR Alarms.Al.Al_MA.Info.Active;
            ELSE
                slavesOk := TRUE;
                FOR i := 1 TO TO_DINT(SlavesNum) DO
                    {IF NOT DEF(MPXONE_BASIC)}
                    slavesOk := slavesOk AND (Slaves[i].myInputRegisters[017] >= TO_UINT(DFR_CHECK_END) OR Slaves[i].myInputRegisters[17] <= TO_UINT(DFR_IDLE) ) OR NOT Slaves[i].Info.IsOnline; // DfrStatus on slaves
                    {ELSE}
                    slavesOk := slavesOk AND (Slaves[i].myInputRegisters[011] >= TO_UINT(DFR_CHECK_END) OR Slaves[i].myInputRegisters[011] <= TO_UINT(DFR_IDLE) ) OR NOT Slaves[i].Info.IsOnline; // DfrStatus on slaves
                    {ENDIF}
                END_FOR;
                // Optionally ignore the sync by parameter
                slavesOk := slavesOk OR NOT DfrMasterEndSync;
            END_IF;

            {IF NOT DEF(MPXONE_BASIC)}
            // Multiplexed valves management
            IF multiplexHotGasType THEN
                // Suction solenoid valve for Multiplexed Hot Gas Defrost
                S_VlvOn := TRUE;
                // Equalizing solenoid valve for Multiplexed Hot Gas Defrost
                E_VlvOn := FALSE;
            ELSE
                S_VlvOn := FALSE;
                E_VlvOn := FALSE;
            END_IF;
            {ENDIF}

            // Clean Dfr temorary vars
            DfrRTRIG(CLK := FALSE);
            //DfrOnTimer := T#0s;
            DfrOnTON(
            	IN := FALSE,
            	PT := T#0s
            );
            DfrOnTON2(
            	IN := FALSE,
            	PT := T#0s
            );
            DfrEndedByTime  := FALSE;
            Dfr2EndedByTime := FALSE;
            MachineTON(IN := FALSE, PT := T#10s); // Reset TIMER

            IF slavesOk THEN
                DfrStatus := DFR_DRIPPING;
                DfrPerformedCntLog := DfrPerformedCntLog + 1;
            END_IF;

        DFR_DRIPPING : //------------- DEFROST DRIPPING STATUS

            DfrCompOff := TRUE;

            {IF NOT DEF(MPXONE_BASIC)}
            // Multiplexed valves management
            IF multiplexHotGasType THEN
                // Suction solenoid valve for Multiplexed Hot Gas Defrost
                S_VlvOn := FALSE;
                // Equalizing solenoid valve for Multiplexed Hot Gas Defrost
                E_VlvOn := TRUE;
            ELSE
                S_VlvOn := FALSE;
                E_VlvOn := FALSE;
            END_IF;
            {ENDIF}

            // Dripping time counter
            MachineTON(IN := TRUE,
                    PT := TO_TIME(TO_UDINT(DripTime) * 1000 * 60));

            IF MachineTON.Q THEN
                DfrStatus := DFR_POST_DRIPPING;
                MachineTON(IN := FALSE, PT := T#10s); // Reset TIMER
            END_IF;

        DFR_POST_DRIPPING : //------------- DEFROST POST DRIPPING STATUS

            // Restart the cooling
            DfrCompOff := FALSE;

            {IF NOT DEF(MPXONE_BASIC)}
            // Multiplexed valves management
            IF multiplexHotGasType THEN
                // Suction solenoid valve for Multiplexed Hot Gas Defrost
                S_VlvOn := TRUE;
                // Equalizing solenoid valve for Multiplexed Hot Gas Defrost
                E_VlvOn := FALSE;
            ELSE
                S_VlvOn := FALSE;
                E_VlvOn := FALSE;
            END_IF;
            {ENDIF}

            // POST Dripping time
            MachineTON(IN := TRUE,
                    PT := TO_TIME(TO_UDINT(PostDripTime) * 1000 * 60));

            IF MachineTON.Q THEN

                DfrStatus := DFR_IDLE;
                ManDfr := FALSE;
                NetworkDfr := FALSE;
                MachineTON(IN := FALSE, PT := T#10s); // Reset TIMER
                CurrentTBisPow := FALSE;
            END_IF;

    END_CASE;

    // Force command on slave devices
    //ForceTON(IN := ForceWrite, PT := T#10s);
    //IF ForceWrite THEN
    //    IF isMaster AND NOT DisNetworkDfr AND SlavesNum > 0 THEN
    //        FOR i := 1 TO TO_DINT(SlavesNum) DO
    //            Slaves[i].myCoilStatus[59] := ForceValue; // ManDfr in BMS table
    //        END_FOR;
    //    END_IF;
    //END_IF;
    //IF ForceTON.Q THEN
    //    ForceWrite := FALSE;
    //END_IF;

END_PROGRAM

END_NAMESPACE

(* ---- 080_FanRegMng.st ---- *)
USING System;
USING Libs.Math;
USING System.Timer;
USING Libs.Hysteresis;

NAMESPACE LibraryNamespaceAndVersion

PROGRAM FanRegMng

    VAR
        FansRegValues : ARRAY [1..2] OF REAL;
        i : INT;
        FansHyst, CutOffHyst : HysterAdv;
        RegVal, tmpReq : REAL;
        FansRegTON, FansPeekTON : TON;
        //FansPeekTOF             : TOF;
        FansStarting            : R_EDGE;
        FansMinOut_tmp          : REAL;
        DelayAfterFirstCycle    : TON;

    END_VAR

     //wait restore default
    IF SW_Update THEN
        RETURN;
    END_IF;

    IF firstCycle THEN
        RETURN;
    END_IF;

    CASE FanMngConfig OF
        0: // Always ON
        FansOn := UnitOn AND NOT WaitForUpdate ;

        1: // Modulating on Sa - Sb

        // Get regulation values
        FOR i := 1 TO 2 DO
            IF FansRegCnf[i] > 0 AND FansRegCnf[i] <= TO_USINT(UPPER_BOUND(RegValues,1)) THEN
                FansRegValues[i] := RegValues[FansRegCnf[i]];
            ELSE
                FansRegValues[i] := 0.0;
            END_IF;
        END_FOR;

        RegVal := FansRegValues[1] - FansRegValues[2];

        2: // Modulating on Sa
        IF FansRegCnf[1] > 0 AND FansRegCnf[1] <= TO_USINT(UPPER_BOUND(RegValues,1)) THEN
            FansRegValues[1] := RegValues[FansRegCnf[1]];
        ELSE
            FansRegValues[1] := 0.0;
        END_IF;
        FansRegValues[2] := 0.0;

        RegVal := FansRegValues[1] - FansRegValues[2];

        3: // Always ON except with door open and DIP configured and active - if DIP is not configured it works as F0 (FanMngConfig) = 0
        FansOn := UnitOn AND NOT WaitForUpdate AND (NOT(Din_Cfg.Fct.DoorOn.Ch > 0 AND DigitalInputs.Fct.DoorOn) OR Din_Cfg.Fct.DoorOn.Ch = 0) ;

    END_CASE;
    {IF NOT DEF(MPXONE_BASIC)}
    FansMinOut_tmp := FansMinOut;
    {ELSE}
    FansMinOut_tmp := 0.0;
    {ENDIF}

    IF UnitOn AND (FanMngConfig > 0 AND FanMngConfig<3) THEN
        FansHyst(In := RegVal, 	SetP := FansSet, DiffLeft := FansDiff, DiffRight := 0.0, Reverse := TRUE);

        FansOn := FansHyst.Out;

        tmpReq := (FansSet - RegVal) / FansDiff * 100;
        // Limit the request
        IF tmpReq < 0 THEN
            tmpReq := 0;
        END_IF;
        IF tmpReq > 100 THEN
            tmpReq := 100;
        END_IF;

        // Cut-Off if FansMinOut is > 0
        CutOffHyst( In := RegVal, SetP := FansCutOff, DiffLeft := 0.0, DiffRight := 1.0, Reverse := FALSE);
    ELSE
        FansMinOut_tmp := 0.0;
        tmpReq := 0.0;
        CutOffHyst( In := 999.9, SetP := FansCutOff, DiffLeft := 0.0, DiffRight := 1.0, Reverse := FALSE);
    END_IF;

    CASE DfrStatus OF
        DFR_IDLE, DFR_CALL:
            IF NOT CntDwnSafT.DevOn AND RegFanConfig AND NOT DfrNatural THEN
                FansOn := FALSE;
                tmpReq := 0.0;
            END_IF;

        DFR_DFR, DFR_CHECK_END:
            IF DfrFanCfg THEN
                FansOn := FALSE;
                tmpReq := 0.0;
                FansMinOut_tmp := 0.0;
            END_IF;

        DFR_DRIPPING:
            FansOn := FALSE;
            tmpReq := 0.0;
            FansMinOut_tmp := 0.0;

        DFR_POST_DRIPPING:
            IF DfrPDFanCfg THEN
                FansOn := FALSE;
                tmpReq := 0.0;
                FansMinOut_tmp := 0.0;
            END_IF;
    END_CASE;

    {IF NOT DEF(MPXONE_BASIC)}
    FansReq := Scaler(tmpReq, 0, 100, FansMinOut_tmp, FansMaxOut);
    {ELSE}
    FansReq := Scaler(tmpReq, 0, 100, FansMinOut_tmp, 100.0);
    {ENDIF}

    // Modulating fan cut-off
    IF CutOffHyst.Out THEN
        FansReq := 0.0;
    END_IF;

    // Periodic or startup speedup

    FansRegTON(IN := FansReq > 0 AND FansSpeedupTime > 0 AND NOT FansRegTON.Q, PT := TO_TIME( TO_DINT(FansSpeedupTime) * 60 * 1000 ));

    IF FansRegTON.Q AND FansPeekTime > 0 THEN
        FansStarting(In := FALSE, Reset := TRUE);
    END_IF;

    FansStarting(In := FansReq > 0 AND FansPeekTime > 0, Reset := FansPeekTON.Q);
    FansPeekTON(IN := FansStarting.Out, PT := TO_TIME(TO_DINT(FansPeekTime) * 1000));

    IF FansStarting.Out THEN
        FansOn := TRUE;
        FansReq := 100.0;
    END_IF;

    // Alarm management
    IF (Alarms.Al.AlExtDin.Info.Active OR (Alarms.Al.AlDelayExtDin.Info.Active AND AlDinDelay>0)) AND RegFanConfig
        //TRAC #111: if AlDinDelay (param.DIb) = 0 --> only warning
        //Fan off if F2 is set as "always off", else fan's behavior depends on F0
            OR GenFctAlarm_Serious THEN //ISSUE #35
        FansOn := FALSE;
        tmpReq := 0;
    END_IF;
    // Issue #22 added exit for UnitOn=False
    IF (DigitalInputs.Fct.DoorOff AND Din_Cfg.fct.DoorOff.Ch <> 0 AND NOT Alarms.Al.Al_Door.Info.Active) OR NOT UnitOn THEN
        FansOn := FALSE;
        FansReq := 0.0;
    END_IF;

    CASE CmdFans OF
        0: // Forced OFF
        FansOn := FALSE;
        FansReq := 0;
        1:
            DelayAfterFirstCycle(IN := TRUE, PT := T#3s);
            CompFanDelay_TON();          //Trac #143 Fan spike on startup with C0>0 (delay on startup) --> recall FB for UPD ET
            IF CompFanDelay_TON.ET > T#0ms  THEN
                FansOn := FALSE;
                FansReq := 0.0;
            END_IF;
        2: // Forced ON
        FansOn := TRUE;
        FansReq := 100;
    END_CASE;

    //Used for ebmpapst fans ESM series - Modbus communication
    SpeedReq_EBM_1 := FansReq * TO_REAL(En_EbmpapstFan_1);

END_PROGRAM

END_NAMESPACE

(* ---- 085_EBM_ESMseriesMng.st ---- *)
USING System.Serial;
USING System.Timer;
USING System;
USING System.Math;
USING System.Util;
USING Libs.EbmpapstFan_Basic;

VAR_GLOBAL
    {ATTRIBUTE UOM PERCENT}
	{METADATA MIN_VAL 0}
	{METADATA MAX_VAL 100}
    SpeedReqPerc_EBM_1 : UINT := 0;

    Ebmpapst_ESM : EbmpapstFan_Basic;
    //Ebmpapst_ESM : EbmpapstFan_Basic;

    SpeedReq_EBM_1          : REAL;
	FW_Reebot_EBM_1         : BOOL;
	LdNewVal_EBM_1          : BOOL;
	ResAlrmInternal_EBM_1   : BOOL;
	Online_EBM_1            : BOOL;
    CtrlModeAct_EBM_1       : UINT;
    CntWorkHrsBkp_EBM_1     : UDINT;
    CurrRotDir_EBM_1        : UINT;
    MotStatus_EBM_1         : MOT_STATUS_EBM_ESM;
    Warn_EBM_1              : WARNING_EBM_ESM;
    ComStatus_EBM_1         : USINT;
    Al_Offline_EBM_1        : BOOL;
    MaxSpeed_EBM_1          : UINT;
    CurrSpeed_EBM_1         :UINT;
    SerNo_EBM_1             : SERIAL_NUM_EBM;
    LdNewAddr_EBM_1         : BOOL;
    NewAddr_EBM_1           : UINT;
END_VAR

VAR_GLOBAL PERSISTENT
    DetectionRange          : TIME := T#2s;
    PollingDelay            : UINT(0..3000) := 50;
    Timeout                 : UINT(200..3000) := 200;
    CommandDelay            : UINT(0..1000) := 20;
    En_EbmpapstFan_1        : BOOL;
    SerInterfaceSet_EBM_1   : CTRL_BOARD_MBM_PARAM_EBM;
    RotDir_EBM_1            : BOOl := TRUE;
    CtrlMode_EBM_1          : USINT := 1;
END_VAR

NAMESPACE LibraryNamespaceAndVersion

PROGRAM EBMMng

    IF NOT firstCycle THEN

        Fieldbus.SerialSettings.Channel := Serial_Channel#FBUS1;
        Fieldbus.SerialSettings.Speed := 19200;
        Fieldbus.SerialSettings.Parity := Serial_Parity#Even;
        Fieldbus.SerialSettings.Stops := SERIAL_STOP_1;

        SerialChangeSettings(Fieldbus.SerialSettings);
    END_IF;

    Fieldbus.Info.DetectionRange := DetectionRange;
    Fieldbus.Info.PollingDelay := PollingDelay;
    Fieldbus.Info.Retry := 5;

    Ebmpapst_ESM(
    	SpeedReq_EBM        := SpeedReq_EBM_1,
    	RotDir_EBM          := RotDir_EBM_1,
    	CtrlMode_EBM        := CtrlMode_EBM_1,
    	SerInterfaceSet_EBM := SerInterfaceSet_EBM_1,
    	FW_Reebot_EBM       := FW_Reebot_EBM_1,
    	LdNewVal_EBM        := LdNewVal_EBM_1,
    	ResAlrmInternal_EBM := ResAlrmInternal_EBM_1,
        LdNewAddr_EBM       := LdNewAddr_EBM_1,
        NewAddr_EBM         := NewAddr_EBM_1,
    	En_EbmpapstFan      := En_EbmpapstFan_1,
    	Online_EBM          => Online_EBM_1,
    	MaxSpeed_EBM        => MaxSpeed_EBM_1,
    	CurrSpeed_EBM       => CurrSpeed_EBM_1,
    	CntWorkHrsBkp_EBM   => CntWorkHrsBkp_EBM_1,
    	CurrRotDir_EBM      => CurrRotDir_EBM_1,
    	SerNo_EBM           => SerNo_EBM_1,
    	MotStatus_EBM       => MotStatus_EBM_1,
    	Warn_EBM            => Warn_EBM_1,
    	Al_Offline_EBM      => Al_Offline_EBM_1
    );

    //Fan 2 offline, increase speed of fan 1 and fan 3
    Alarms.Al.EBM1_Offline.Info.Trigger := Al_Offline_EBM_1;

END_PROGRAM

END_NAMESPACE

(* ---- 090_ExvMng.st ---- *)
{IF NOT DEF(MPXONE_BASIC)}
USING Libs.EVD_ACU;
USING Libs.MPXone_Smoothlines;
USING System;
USING Libs.Logics;
USING Libs.Math;
USING System.Math;
USING System.Timer;
USING Libs.Hysteresis;
USING Libs.SignalGeneration;
{ENDIF}

// Use shared pressure probe and EVD regulation
{IF NOT DEF(MPXONE_BASIC)}
VAR_GLOBAL
    MachineVars: Libs.EVD_ACU.MACHINE_DATA_VARS;
    MachineParams : Libs.EVD_ACU.MACHINE_DATA_PARAMS;

    {IF NOT DEF(MPXONE_ADVANCED)}
    MachineDrivingExtPosit      : MAIN_MachineDrivingExtPosit;
    ExtPosit_EVD                : System.EVD.TEEV;
	DevErr                      : UINT;
	DevErr_EVD                  : INT;
    ErrCode_EVD                 : INT;

    {IF NOT DEF(MPXONE_BASIC)}
    EvdMpxReg                   : Libs.EvdMPX.EvdMPXReg;
    {ENDIF}

	OfflineAlrm_EVD             : BOOL;
    Online_EVD                  : BOOL;
    CfgErr_EVD                  : UINT;
    {ENDIF}

END_VAR
{ENDIF}

{IF NOT DEF(MPXONE_BASIC)}

{IF NOT DEF(MPXONE_ADVANCED)}
VAR_GLOBAL PERSISTENT
	EVD_MB_CmdDelay : UINT(0..1000)             := 5;
    EVD_MB_Timeout : UINT(200..3000)            := 500;
    EVD_MB_DetectionTimeOut : UINT(200..5000)   := 500;
END_VAR
{ENDIF}

NAMESPACE LibraryNamespaceAndVersion

PROGRAM ExvMng

    VAR
        MachineInit                 : MAIN_MachineInit;
        MachineServiceTimerUpdate   : MAIN_MachineServiceTimerUpdate;
        MachineCanGo                : MAIN_EVDCanGoMng;
        MachineController           : MAIN_MachineController;
        {IF DEF(MPXONE_ADVANCED)}
        MachineDriving              : MAIN_MachineDriving;
        {ENDIF}

        EVDCanGo                    : BOOL := TRUE;
        Ts                          : UDINT := 300;

        ShOffset : REAL;
        GetMPXoneSmLine : MPXone_Smoothlines;
//        ShSetPID : PID_Incr;

        AfterDfrTON : TON;
        AfterDfrFEDGE : F_EDGE;

        ManPar : RF_Trig;

        BlockAlarmTON: TON;
        ExvVlvBlockChk : BOOL;
        VlvBlockHiHyst, VlvBlockLowHyst : HysterAdv;

        SuctTDutyCycle : BlinkOnOff;
        SuctTDutyFEDGE : F_TRIG;
        Sm_VirtualPrb_PrevVal : REAL;
    END_VAR

    VAR_TEMP
        tmp_CoolingCapacity : UINT;
    END_VAR

    //wait restore default
    IF SW_Update THEN
        RETURN;
    END_IF;

    VlvPresent := ValveCnf > 0 AND (isMedium OR isAdvanced);

    IF VlvPresent THEN
        {REGION PARAMETERS}
            //ExvPIDKp_checkWoC(val_In1 := ExvKp, val_In2 := MachineParams.Engine_params.PID_PARAMS.Kp);
            //ExvPIDTi_checkWoC(val_In1 := MachineParams.Engine_params.PID_PARAMS.Ti, val_In2 := );

            MachineParams.Engine_params.PID_PARAMS.Kp := ExvKp;
            MachineParams.Engine_params.PID_PARAMS.Ti := TO_REAL(ExvTi);
            MachineParams.Engine_params.PID_PARAMS.Td := TO_REAL(ExvTd);

            // Low SH settings
            MachineParams.SH_params.SHProtection_params.LowSHAlarmDelay := LowSH_AlrmDelay;
            MachineParams.SH_params.SHProtection_params.LowSHThreshold := LowSH_Thrsh;
            MachineParams.SH_params.SHProtection_params.LowSHTi := LowSH_Ti;

            // Low suction temperature settings
            MachineParams.SH_params.SHProtection_params.LowSuctAlarmDelay := LowSuctAlrmDelay;
            MachineParams.SH_params.SHProtection_params.LowSuctThreshold := LowSuctThrsh;

            // MOP settings
            MachineParams.SH_params.SHProtection_params.MOPAlarmDelay := MOP_AlrmDelay;
            MachineParams.SH_params.SHProtection_params.MOPSuctionTemperatureThreshold := MOP_SuctTempThrsh;
            MachineParams.SH_params.SHProtection_params.MOPThreshold := MOP_Thrsh;
            MachineParams.SH_params.SHProtection_params.MOPTi := MOP_Ti;

            // LOP settings
            MachineParams.SH_params.SHProtection_params.LOPAlarmDelay := TO_UINT(LOP_AlrmDelay);
            MachineParams.SH_params.SHProtection_params.LOPThreshold := LOP_Thrsh;
            MachineParams.SH_params.SHProtection_params.LOPTi := LOP_Ti;

            // Start of valve regulation
            MachineParams.Engine_params.StartEEVOpenRatio := TO_UINT(StartEEVOpenRatio);
            MachineParams.Engine_params.RegulationStartDelay := 0;

        {ENDREGION }

        {REGION CALCULATE_SH_SETPOINT}
        GetMPXoneSmLine(
        	VirtualProbe_SL          := VirtualProbe,
        	TempSetP_SL              := TempSetP,
        	TempDiff_SL              := TempDiff,
        	SmLineKp_SL              := SmLineKp,
        	SmLineTi_SL              := SmLineTi,
        	SmLineTd_SL              := SmLineTd,
        	SmLineSHOffset_SL        := SmLineSHOffset,
        	EnSmoothLine_SL          := EnSmoothLine,
        	SmLine_SH_thrsh_SL       := SmLine_SH_thrsh,
        	ShOffset_SL              => ShOffset,
        	Sm_VirtualPrb_PrevVal_SL := Sm_VirtualPrb_PrevVal
        );

        ActualShSetP := SHSetP + ShOffset;

        BMS_SHSet := ActualShSetP;

        MachineParams.SH_params.SHset := SHSetP;
        {ENDREGION }

        {REGION EVD_ACU_CORE}

        (*cooling capacity sent to valve*)
        // P10 management
        tmp_CoolingCapacity := 100 - (99 * TO_UINT(Alarms.Al.Al_LSA.Info.Trigger OR Alarms.Al.Al_LSH.info.Trigger)); // TRAC #133 removed check on ExvEnCloseLsa (P10), EXV has to close independently

        // PM5 management
        IF tmp_CoolingCapacity > 1 THEN
            tmp_CoolingCapacity := 100 - (99 * TO_UINT(ExvEnCloseMOP AND Alarms.Al.Al_MOP.Info.Trigger));
        END_IF;

        IF tmp_CoolingCapacity < 100 THEN
            {IF NOT DEF (MPXONE_BASIC)}
                MachineVars.Engine_vars.UnitPower := 10; //close o valve during Alarm; not set=0 otherwise Alarm aren't check by EVD_ACU lib
            {ENDIF}
        ELSE
            IF isMaster AND MstVlvConfig THEN
                MachineVars.Engine_vars.UnitPower := 100 * TO_UINT(MstTempRegStatus AND (DfrStatus = DFR_IDLE OR DfrStatus = DFR_POST_DRIPPING));
            ELSE
                MachineVars.Engine_vars.UnitPower := 100 * TO_UINT(TempRegStatus AND (DfrStatus = DFR_IDLE OR DfrStatus = DFR_POST_DRIPPING));
            END_IF;
        END_IF;

        (*EXV works on suction superheat*)
        IF ValveCnf = 1 OR ValveCnf = 2 OR (ValveCnf = 6 AND VlvPressPrbTyp = 14) THEN
            MachineVars.SH_vars.EvaporationTemperature := EvapSatTemp;
        ELSE
            EvapSatTemp := MachineVars.SH_vars.EvaporationTemperature;
        END_IF;

        MachineVars.SH_vars.SuctionTemperature := AnalogInputs.Fct.SuctT - ShOffset;

        // During defrost force the valve status if needed
        IF DfrStatus = DFR_DFR THEN
            CASE DfrVlvPos OF

                2..100: // fixed % if configured
                MachineVars.ManualPositioner_vars.ManualPositioningEnable := TRUE;
                MachineVars.ManualPositioner_vars.ManualPositionSteps := TO_UINT(TO_REAL(DfrVlvPos) / 100.0 * 480.0);

                1: // Keep the valve closed during defrost
                MachineVars.ManualPositioner_vars.ManualPositioningEnable := TRUE;
                MachineVars.ManualPositioner_vars.ManualPositionSteps := 0;

                0: // Default mng (Normal regulation)
                MachineVars.ManualPositioner_vars.ManualPositioningEnable := FALSE;
                MachineVars.ManualPositioner_vars.ManualPositionSteps := 0;

            END_CASE;
        /*ELSE
            MachineVars.ManualPositioner_vars.ManualPositioningEnable := FALSE;
            MachineVars.ManualPositioner_vars.ManualPositionSteps := 0;*/
        END_IF;

        IF DfrStatus = DFR_DRIPPING THEN
            MachineVars.ManualPositioner_vars.ManualPositioningEnable := TRUE;
            MachineVars.ManualPositioner_vars.ManualPositionSteps := 0;
        END_IF;

        // After the defrost keep the valve opening for Pdd time
        AfterDfrFEDGE( In := DfrStatus = DFR_DRIPPING, Reset := AfterDfrTON.Q);
        AfterDfrTON( IN := AfterDfrFEDGE.Out, PT := TO_TIME(TO_UDINT(ExvDelayDfr) * 60 * 1000));
        IF AfterDfrFEDGE.Out AND NOT AfterDfrTON.Q THEN
            MachineVars.ManualPositioner_vars.ManualPositioningEnable := TRUE;
            MachineVars.ManualPositioner_vars.ManualPositionSteps := TO_UINT(TO_REAL(StartEEVOpenRatio) / 100.0 * 480.0);
        END_IF;
        IF AfterDfrTON.Q THEN
            MachineVars.ManualPositioner_vars.ManualPositioningEnable := FALSE;
            MachineVars.ManualPositioner_vars.ManualPositionSteps := 0;
        END_IF;

        IF DfrType = 1 OR DfrType = 3 THEN
            MachineVars.Engine_vars.UnitPower := 100 * TO_UINT(TempRegStatus AND ( DfrStatus <> DFR_POST_DRIPPING ));
        END_IF;

        (* Duty cycle in case of SuctT sensor broken *)
        SuctTDutyFEDGE(CLK := SuctTBroken);
        IF SuctTBroken THEN
            //Duty cycle 2 min at 0.5*cP1 (prepositioning) and 1 min at Psb (stand-by position)
            MachineVars.ManualPositioner_vars.ManualPositioningEnable := TRUE;
            SuctTDutyCycle(In := SuctTBroken, T_On := 120, T_Off := 60);
            IF SuctTDutyCycle.Out THEN
                MachineVars.ManualPositioner_vars.ManualPositionSteps := TO_UINT(0.5*(TO_REAL(StartEEVOpenRatio) / 100.0 * 480.0));
            ELSE
                MachineVars.ManualPositioner_vars.ManualPositionSteps := StandbyEEVOpenPosition;
            END_IF;
        ELSIF SuctTDutyFEDGE.Q THEN
            MachineVars.ManualPositioner_vars.ManualPositioningEnable := FALSE;
            MachineVars.ManualPositioner_vars.ManualPositionSteps := 0;
        END_IF;

        // Manual management from SPV, APP or parameters
        ManPar(CLK := EnManExv OR Alarms.Al.Al_LSA.Info.Trigger);
        IF ManPar.Q OR EnManExv THEN
            MachineVars.ManualPositioner_vars.ManualPositioningEnable   := EnManExv OR Alarms.Al.Al_LSA.Info.Trigger;
            IF Alarms.Al.Al_LSA.Info.Trigger THEN
                 // LSA Force clousure of valve by manpos
                MachineVars.ManualPositioner_vars.ManualPositionSteps       := 0;
            ELSE
                MachineVars.ManualPositioner_vars.ManualPositionSteps       := PosManExv;
            END_IF;
        END_IF;
                    // reset manul forcinng to allow reset of alarm same differential done in EVD_ACU lib)
        IF Alarms.Al.Al_LSA.Info.Trigger  AND AnalogInputs.Fct.SuctT >  LowSuctThrsh + 3 THEN
            MachineVars.ManualPositioner_vars.ManualPositioningEnable   := FALSE;
        END_IF;

        MachineInit(MachineParams := MachineParams, MachineVars := MachineVars);
        MachineServiceTimerUpdate( MachineVars := MachineVars );

        MachineCanGo(
                RegulationType := 6,
                Machine_params := MachineParams,
                Machine_vars := MachineVars,
                EVDCanGo := EVDCanGo
                );

        MachineController(MachineParams := MachineParams, MachineVars := MachineVars, Ts := Ts);

    END_IF;

    ActualSH := AnalogInputs.Fct.SuctT - EvapSatTemp;

    {IF DEF(MPXONE_ADVANCED)}
    IF PwrSupplyFailure THEN // Manage the valve closure in case of power failure
        EVDCanGo := FALSE;
        MachineVars.Engine_Vars.EEV_Vars.FastClosingSpeedEnable := 1;

        // If the power comes back restore the regulation
            IF  (u[9].r > 0 AND ExvVlvPosition < 1) THEN //u[9]>0 means that the power supply is present (230Vac)
            PwrSupplyFailure := FALSE;
            MachineVars.Engine_Vars.EEV_Vars.FastClosingSpeedEnable := 0;
            EVDCanGo := TRUE;
        END_IF;

    END_IF;

    MachineDriving( ID_Driver := 1,
        MachineVars := MachineVars,
        MachineParams := MachineParams);
    {ENDIF}
    {IF NOT DEF(MPXONE_ADVANCED)}
    MachineDrivingExtPosit(
        ExtPosit_CPCOE  := ExtPosit_EVD,
        MachineVars     := MachineVars,
        MachineParams   := MachineParams
    );
    {ENDIF}
    {ENDREGION }

    {REGION EVD_MPX}
    {IF NOT DEF(MPXONE_ADVANCED)}

    //EVDice and EVDmini management
    EvdMpxReg(
        DevAddr_EVD := EvdAddr,
        En_EVD := (ValveCnf = 2 OR ValveCnf = 6) AND EVDCanGo,
        GasIndex := RfrgTyp,

        Online_EVD => Online_EVD,
        OfflineAlrm_EVD => OfflineAlrm_EVD,
        DevErr => DevErr_EVD,
        ErrCode => ErrCode_EVD,
        CfgErr_EVD => CfgErr_EVD,
        EVD_EvapP => EVD_EvapP,

        Al_S1Probe => Alarms.Al.AL_DA1_EVDmini.Info.Trigger,
        Al_S2Probe => Alarms.Al.AL_DA2_EVDmini.Info.Trigger,
        Al_EEprom_EVD => Alarms.Al.Al_DEE_EVDmini.Info.Trigger,
        Al_EmergencyClosing => Alarms.Al.Al_DE5_EVDmini.Info.Trigger,

        MachineVars := MachineVars,
        MachineParams := MachineParams,
        ExtPosit_EVD := ExtPosit_EVD,
        EVD_Digin1Cfg := EVD_Digin1Cfg,
        //VAR_IN_OUT CONSTANT
        VlvPressPrbTyp := VlvPressPrbTyp,
        EvaporationPressure := AnalogInputs.Fct.EvapP,
        SmoothLineOffset := ShOffset,
        ValveCnf := ValveCnf,
        MB_Timeout          := EVD_MB_Timeout,
    	MB_CmdDelay         := EVD_MB_CmdDelay,
        MB_DetectionTimeout := EVD_MB_DetectionTimeOut
    );
     Alarms.Al.Warn_EVD_Fw.Info.Trigger := CfgErr_EVD > 0;
    {ENDIF}
    {ENDREGION }

    IF MachineVars.Engine_vars.EEV_vars.CurrentEstimatedPosition > 1 THEN
        ExvVlvPosition := TO_USINT( TO_REAL(MachineVars.Engine_vars.EEV_vars.CurrentEstimatedPosition) / 4.8 );
    ELSE
        ExvVlvPosition := 0;
    END_IF;

    IF ExvVlvPosition > 100 THEN
        ExvVlvPosition := 100;
    END_IF;

    // check valve blocked conditions
    VlvBlockHiHyst(In := ActualSH, SetP := ActualShSetp, DiffLeft := 0.0, DiffRight := 0.5, Reverse := FALSE);
    VlvBlockLowHyst(In := ActualSH, SetP := ActualShSetp, DiffLeft := 0.5, DiffRight := 0.0, Reverse := TRUE);

    ExvVlvBlockChk := (ExvVlvPosition >= 90 AND VlvBlockHiHyst.Out) OR (ExvVlvPosition <= 10 AND VlvBlockLowHyst.Out);
    BlockAlarmTON(IN := NOT EnManExv AND EnBloAlarm AND ExvVlvBlockChk, PT := T#25m);//check condition valve blocked ('bLO') too open or too closed

    {REGION ALARMS_MNG}

    IF ValveCnf = 1 OR ValveCnf = 2 OR ValveCnf = 5 THEN
        Alarms.Al.Al_LSH.Info.Trigger := MachineController.Al_LowSH;
        Alarms.Al.Al_LOP.Info.Trigger := MachineController.Al_LOP;
        Alarms.Al.Al_MOP.Info.Trigger := MachineController.Al_MOP;
        Alarms.Al.Al_LSA.Info.Trigger := MachineController.Al_LowSuct;

    {IF NOT DEF(MPXONE_ADVANCED)}
    ELSIF ValveCnf = 6 THEN
        Alarms.Al.Al_LSH.Info.Trigger := EvdMpxReg.Al_LowSH;
        Alarms.Al.Al_LOP.Info.Trigger := EvdMpxReg.Al_LOP;
        Alarms.Al.Al_MOP.Info.Trigger := EvdMpxReg.Al_MOP;
        Alarms.Al.Al_LSA.Info.Trigger := EvdMpxReg.Al_LowSuct;
    {ENDIF}
    END_IF;

    Alarms.Al.Al_bLO.Info.Trigger := BlockAlarmTON.Q AND ValveCnf > 0;

    {IF NOT DEF(MPXONE_ADVANCED)}
    Alarms.Al.Al_Edc.Info.Trigger := NOT Online_EVD AND (ValveCnf = 2 OR ValveCnf = 5 OR ValveCnf = 6);
    {ENDIF}
    {ENDREGION}

END_PROGRAM

FUNCTION_BLOCK checkWriteOnChange_REAL
    VAR_IN_OUT
        val_In1, val_In2 : REAL;
    END_VAR

    VAR
        changeByIn1, changeByIn2 : BOOL;
        prevVal_In1, prevValIn2 : REAL;
    END_VAR

    IF val_In1 <> prevVal_In1 THEN
        prevVal_In1 := val_In1;
        changeByIn1 := TRUE;
    END_IF;

    IF val_In2 <> prevValIn2 THEN
        prevValIn2 := val_In2;
        changeByIn2 := TRUE;
    END_IF;

    IF changeByIn1 THEN val_In2 := val_In1; END_IF;

    IF changeByIn2 THEN val_In1 := val_In2; END_IF;

END_FUNCTION_BLOCK
{ENDIF}

END_NAMESPACE

(* ---- 100_HeatersMng.st ---- *)
USING Libs.PID_Incr;
USING System.Timer;
USING System;
USING Libs.Hysteresis;

NAMESPACE LibraryNamespaceAndVersion

PROGRAM HeatersMng
    VAR
        HeatersPID : PID_Incr;

        ActiveTON, PeriodTON : TON;
        ActiveTIME, PeriodTIME : TIME;

        MinOut, MaxOut, SafeKP : REAL;

        Ti_RailHeaters : UINT;

        {ATTRIBUTE UOM CELSIUS}
        CutOff : REAL;
        CutOffHyst : HysterAdv;
    END_VAR

    VAR_TEMP
        ManModePID_en : BOOL;
        ManModePID_val : REAL;
    END_VAR

    //wait restore default
    IF SW_Update THEN
        RETURN;
    END_IF;

    IF firstCycle THEN
        RETURN;
    END_IF;

    IF UnitOn THEN
        MaxOut := 100.0;
        MinOut := 10.0;
        CutOff := 5.0;

        // Avoid division by Zero
        IF HeatersDiff > 0 THEN

            IF Ain_Cfg.Fct.GlassT.ch <> 0 THEN
                Ti_RailHeaters := 600;
            ELSE
                Ti_RailHeaters := 0;
            END_IF;

            SafeKP := (MaxOut - MinOut) / HeatersDiff;

//            HeatersPID(RegVar_PID_Incr := Probes.Prb.GlassT, SetP_PID_Incr := Probes.Prb.DewPoint + HeaterOffs,
//                DeadBand_PID_Incr := 0.0, Kp_PID_Incr := SafeKP, Ti_PID_Incr := Ti_RailHeaters, Td_PID_Incr := 0,
//                LowLim_PID_Incr := MinOut, HighLim_PID_Incr := MaxOut, Period_PID_Incr := 500, CoolHeatMode_PID_Incr := TRUE,
//                RevMode_PID_Incr := FALSE, ManModeVal_PID_Incr := 100.0, En_ManMode_PID_Incr := Probes.Prb.GlassT <= Probes.Prb.DewPoint + HeaterOffs,
//                En_PID_Incr := TRUE);

            IF AnalogInputs.Fct.GlassT <= AnalogInputs.Fct.DewPoint + HeaterOffs THEN
                ManModePID_en := TRUE;
                ManModePID_val := 100.0;
            ELSIF (AnalogInputs.Fct.GlassT >= AnalogInputs.Fct.DewPoint + HeaterOffs + HeatersDiff) AND
                    (AnalogInputs.Fct.GlassT <= AnalogInputs.Fct.DewPoint + HeaterOffs + HeatersDiff + 5) THEN
                ManModePID_en := TRUE;
                ManModePID_val := 10.0;
            ELSE
                ManModePID_en := FALSE;
            END_IF;

            HeatersPID(RegVar_PID_Incr := AnalogInputs.Fct.GlassT, SetP_PID_Incr := AnalogInputs.Fct.DewPoint + HeaterOffs,
                DeadBand_PID_Incr := 0.0, Kp_PID_Incr := SafeKP, Ti_PID_Incr := Ti_RailHeaters, Td_PID_Incr := 0,
                LowLim_PID_Incr := MinOut, HighLim_PID_Incr := MaxOut, Period_PID_Incr := 500, CoolHeatMode_PID_Incr := FALSE,
                RevMode_PID_Incr := TRUE, ManModeVal_PID_Incr := ManModePID_val, En_ManMode_PID_Incr := ManModePID_en,
                En_PID_Incr := TRUE);

            HeatersOut := TO_USINT(HeatersPID.Req_PID_Incr);

            CutOffHyst(
                In        := AnalogInputs.Fct.GlassT,
            	SetP      := AnalogInputs.Fct.DewPoint + HeaterOffs + HeatersDiff + CutOff,
            	DiffLeft  := 1.0,
            	DiffRight := 0.0,
            	Reverse   := TRUE
            );

            IF NOT CutOffHyst.Out THEN
                HeatersOut := 0;
            END_IF;
        ELSE

            ActiveTIME := TO_TIME(TO_REAL(TO_DINT(ManHeaterPeriod) * 1000 * 60) * TO_REAL(ManHeaterPerc) / 100.0);
            ActiveTON(IN := NOT PeriodTON.Q, PT := ActiveTIME);
            PeriodTIME := TO_TIME(TO_DINT(ManHeaterPeriod) * 1000 * 60);
            PeriodTON(IN := NOT PeriodTON.Q, PT := PeriodTIME);

            IF NOT ActiveTON.Q THEN
                HeatersOut := 100;
            ELSE
                HeatersOut := 0;
            END_IF;
//            SafeKP := 999;
        END_IF;
    ELSE
        // Turn OFF
        HeatersOut := 0;
    END_IF;
END_PROGRAM

END_NAMESPACE
